gfCNCPoint5[12058] = {X 116.0973, Y 79.9611, Z -7.1667, A 0.000, B 0.000, C 0.000 }
gfCNCPoint5[12059] = {X 117.8219, Y 79.1683, Z -7.1667, A 0.000, B 0.000, C 0.000 }
gfCNCPoint5[12060] = {X 119.6162, Y 78.5490, Z -7.1667, A 0.000, B 0.000, C 0.000 }
gfCNCPoint5[12061] = {X 137.8560, Y 58.5204, Z -7.1667, A 0.000, B 0.000, C 0.000 }
gfCNCPoint5[12062] = {X 136.5214, Y 57.9299, Z -7.1667, A 0.000, B 0.000, C 0.000 }
gfCNCPoint5[12063] = {X 135.2529, Y 57.2081, Z -7.1667, A 0.000, B 0.000, C 0.000 }
gfCNCPoint5[12064] = {X 134.0093, Y 56.3192, Z -7.1667, A 0.000, B 0.000, C 0.000 }
gfCNCPoint5[12065] = {X 132.8663, Y 55.3040, Z -7.1667, A 0.000, B 0.000, C 0.000 }
gfCNCPoint5[12066] = {X 131.8367, Y 54.1741, Z -7.1667, A 0.000, B 0.000, C 0.000 }
gfCNCPoint5[12067] = {X 130.9319, Y 52.9419, Z -7.1667, A 0.000, B 0.000, C 0.000 }
gfCNCPoint5[12068] = {X 130.2147, Y 51.7225, Z -7.1667, A 0.000, B 0.000, C 0.000 }
gfCNCPoint5[12069] = {X 129.6199, Y 50.4390, Z -7.1667, A 0.000, B 0.000, C 0.000 }
gfCNCPoint5[12070] = {X 129.1532, Y 49.1035, Z -7.1667, A 0.000, B 0.000, C 0.000 }
gfCNCPoint5[12071] = {X 128.6036, Y 50.3877, Z -7.1667, A 0.000, B 0.000, C 0.000 }
gfCNCPoint5[12072] = {X 127.9093, Y 51.5998, Z -7.1667, A 0.000, B 0.000, C 0.000 }
gfCNCPoint5[12073] = {X 127.0798, Y 52.7237, Z -7.1667, A 0.000, B 0.000, C 0.000 }
gfCNCPoint5[12074] = {X 126.0417, Y 53.8239, Z -7.1667, A 0.000, B 0.000, C 0.000 }
gfCNCPoint5[12075] = {X 124.8743, Y 54.7858, Z -7.1667, A 0.000, B 0.000, C 0.000 }
gfCNCPoint5[12076] = {X 123.5958, Y 55.5942, Z -7.1667, A 0.000, B 0.000, C 0.000 }
gfCNCPoint5[12077] = {X 122.2263, Y 56.2365, Z -7.1667, A 0.000, B 0.000, C 0.000 }
gfCNCPoint5[12078] = {X 120.7872, Y 56.7027, Z -7.1667, A 0.000, B 0.000, C 0.000 }
gfCNCPoint5[12079] = {X 119.3012, Y 56.9853, Z -7.1667, A 0.000, B 0.000, C 0.000 }
gfCNCPoint5[12080] = {X 117.7916, Y 57.0800, Z -7.1667, A 0.000, B 0.000, C 0.000 }
gfCNCPoint5[12081] = {X 111.9185, Y 57.0800, Z -7.1667, A 0.000, B 0.000, C 0.000 }
gfCNCPoint5[12082] = {X 111.7011, Y 57.0780, Z -7.1667, A 0.000, B 0.000, C 0.000 }
gfCNCPoint5[12083] = {X 111.4838, Y 57.0722, Z -7.1667, A 0.000, B 0.000, C 0.000 }
gfCNCPoint5[12084] = {X 111.5702, Y 54.6737, Z -7.1667, A 0.000, B 0.000, C 0.000 }
gfCNCPoint5[12085] = {X 110.3801, Y 54.5570, Z -7.1667, A 0.000, B 0.000, C 0.000 }
gfCNCPoint5[12086] = {X 109.2135, Y 54.2944, Z -7.1667, A 0.000, B 0.000, C 0.000 }
gfCNCPoint5[12087] = {X 108.0882, Y 53.8899, Z -7.1667, A 0.000, B 0.000, C 0.000 }
gfCNCPoint5[12088] = {X 107.0213, Y 53.3498, Z -7.1667, A 0.000, B 0.000, C 0.000 }
gfCNCPoint5[12089] = {X 106.6480, Y 53.5578, Z -7.1667, A 0.000, B 0.000, C 0.000 }
gfCNCPoint5[12090] = {X 106.2658, Y 53.7492, Z -7.1667, A 0.000, B 0.000, C 0.000 }
gfCNCPoint5[12091] = {X 105.0149, Y 54.2383, Z -7.1667, A 0.000, B 0.000, C 0.000 }
gfCNCPoint5[12092] = {X 103.7084, Y 54.5495, Z -7.1667, A 0.000, B 0.000, C 0.000 }
gfCNCPoint5[12093] = {X 102.3713, Y 54.6768, Z -7.1667, A 0.000, B 0.000, C 0.000 }
gfCNCPoint5[12094] = {X 101.0295, Y 54.6179, Z -7.1667, A 0.000, B 0.000, C 0.000 }
gfCNCPoint5[12095] = {X 99.7088, Y 54.3738, Z -7.1667, A 0.000, B 0.000, C 0.000 }
gfCNCPoint5[12096] = {X 98.4345, Y 53.9493, Z -7.1667, A 0.000, B 0.000, C 0.000 }
gfCNCPoint5[12097] = {X 97.2313, Y 53.3524, Z -7.1667, A 0.000, B 0.000, C 0.000 }
gfCNCPoint5[12098] = {X 96.0852, Y 53.9255, Z -7.1667, A 0.000, B 0.000, C 0.000 }
gfCNCPoint5[12099] = {X 94.8734, Y 54.3422, Z -7.1667, A 0.000, B 0.000, C 0.000 }
gfCNCPoint5[12100] = {X 93.6172, Y 54.5952, Z -7.1667, A 0.000, B 0.000, C 0.000 }
gfCNCPoint5[12101] = {X 92.3385, Y 54.6800, Z -7.1667, A 0.000, B 0.000, C 0.000 }
gfCNCPoint5[12102] = {X 85.8951, Y 54.6800, Z -7.1667, A 0.000, B 0.000, C 0.000 }
gfCNCPoint5[12103] = {X 84.6159, Y 54.5951, Z -7.1667, A 0.000, B 0.000, C 0.000 }
gfCNCPoint5[12104] = {X 83.3592, Y 54.3419, Z -7.1667, A 0.000, B 0.000, C 0.000 }
gfCNCPoint5[12105] = {X 82.1469, Y 53.9249, Z -7.1667, A 0.000, B 0.000, C 0.000 }
gfCNCPoint5[12106] = {X 81.0644, Y 55.1572, Z -7.1667, A 0.000, B 0.000, C 0.000 }
gfCNCPoint5[12107] = {X 79.8495, Y 56.2591, Z -7.1667, A 0.000, B 0.000, C 0.000 }
gfCNCPoint5[12108] = {X 78.5178, Y 57.2166, Z -7.1667, A 0.000, B 0.000, C 0.000 }
gfCNCPoint5[12109] = {X 77.0863, Y 58.0174, Z -7.1667, A 0.000, B 0.000, C 0.000 }
gfCNCPoint5[12110] = {X 75.5734, Y 58.6511, Z -7.1667, A 0.000, B 0.000, C 0.000 }
gfCNCPoint5[12111] = {X 73.9986, Y 59.1096, Z -7.1667, A 0.000, B 0.000, C 0.000 }
gfCNCPoint5[12112] = {X 72.3820, Y 59.3871, Z -7.1667, A 0.000, B 0.000, C 0.000 }
gfCNCPoint5[12113] = {X 70.7445, Y 59.4800, Z -7.1667, A 0.000, B 0.000, C 0.000 }
gfCNCPoint5[12114] = {X 64.1851, Y 59.4800, Z -7.1667, A 0.000, B 0.000, C 0.000 }
gfCNCPoint5[12115] = {X 62.4203, Y 59.3720, Z -7.1667, A 0.000, B 0.000, C 0.000 }
gfCNCPoint5[12116] = {X 60.6818, Y 59.0498, Z -7.1667, A 0.000, B 0.000, C 0.000 }
gfCNCPoint5[12117] = {X 58.9955, Y 58.5181, Z -7.1667, A 0.000, B 0.000, C 0.000 }
gfCNCPoint5[12118] = {X 57.3866, Y 57.7848, Z -7.1667, A 0.000, B 0.000, C 0.000 }
gfCNCPoint5[12119] = {X 55.8790, Y 56.8608, Z -7.1667, A 0.000, B 0.000, C 0.000 }
gfCNCPoint5[12120] = {X 54.3715, Y 57.7848, Z -7.1667, A 0.000, B 0.000, C 0.000 }
gfCNCPoint5[12121] = {X 52.7626, Y 58.5181, Z -7.1667, A 0.000, B 0.000, C 0.000 }
gfCNCPoint5[12122] = {X 51.0763, Y 59.0498, Z -7.1667, A 0.000, B 0.000, C 0.000 }
gfCNCPoint5[12123] = {X 49.3378, Y 59.3720, Z -7.1667, A 0.000, B 0.000, C 0.000 }
gfCNCPoint5[12124] = {X 47.5729, Y 59.4800, Z -7.1667, A 0.000, B 0.000, C 0.000 }
gfCNCPoint5[12125] = {X 40.6393, Y 59.4800, Z -7.1667, A 0.000, B 0.000, C 0.000 }
gfCNCPoint5[12126] = {X 38.9799, Y 59.3846, Z -7.1667, A 0.000, B 0.000, C 0.000 }
gfCNCPoint5[12127] = {X 37.3423, Y 59.0996, Z -7.1667, A 0.000, B 0.000, C 0.000 }
gfCNCPoint5[12128] = {X 35.7482, Y 58.6289, Z -7.1667, A 0.000, B 0.000, C 0.000 }
gfCNCPoint5[12129] = {X 34.0334, Y 59.4877, Z -7.1667, A 0.000, B 0.000, C 0.000 }
gfCNCPoint5[12130] = {X 32.2400, Y 60.1674, Z -7.1667, A 0.000, B 0.000, C 0.000 }
gfCNCPoint5[12131] = {X 30.3868, Y 60.6610, Z -7.1667, A 0.000, B 0.000, C 0.000 }
gfCNCPoint5[12132] = {X 28.4929, Y 60.9633, Z -7.1667, A 0.000, B 0.000, C 0.000 }
gfCNCPoint5[12133] = {X 26.3340, Y 61.8578, Z -7.1667, A 0.000, B 0.000, C 0.000 }
gfCNCPoint5[12134] = {X 24.1304, Y 62.6356, Z -7.1667, A 0.000, B 0.000, C 0.000 }
gfCNCPoint5[12135] = {X 21.7252, Y 63.3378, Z -7.1667, A 0.000, B 0.000, C 0.000 }
gfCNCPoint5[12136] = {X 19.2782, Y 63.8767, Z -7.1667, A 0.000, B 0.000, C 0.000 }
gfCNCPoint5[12137] = {X 16.8005, Y 64.2498, Z -7.1667, A 0.000, B 0.000, C 0.000 }
gfCNCPoint5[12138] = {X 14.3033, Y 64.4554, Z -7.1667, A 0.000, B 0.000, C 0.000 }
gfCNCPoint5[12139] = {X 14.3033, Y 85.6951, Z -7.1667, A 0.000, B 0.000, C 0.000 }
gfCNCPoint5[12140] = {X 112.5225, Y 85.6951, Z -7.1667, A 0.000, B 0.000, C 0.000 }
gfCNCPoint5[12141] = {X 113.9417, Y 84.3100, Z -7.1667, A 0.000, B 0.000, C 0.000 }
gfCNCPoint5[12142] = {X 115.5135, Y 83.1008, Z -7.1667, A 0.000, B 0.000, C 0.000 }
gfCNCPoint5[12143] = {X 117.2162, Y 82.0843, Z -7.1667, A 0.000, B 0.000, C 0.000 }
gfCNCPoint5[12144] = {X 119.0264, Y 81.2746, Z -7.1667, A 0.000, B 0.000, C 0.000 }
gfCNCPoint5[12145] = {X 120.9191, Y 80.6827, Z -7.1667, A 0.000, B 0.000, C 0.000 }
gfCNCPoint5[12146] = {X 142.4280, Y 57.0645, Z -7.1667, A 0.000, B 0.000, C 0.000 }
gfCNCPoint5[12147] = {X 141.1651, Y 56.9337, Z -7.1667, A 0.000, B 0.000, C 0.000 }
gfCNCPoint5[12148] = {X 139.9229, Y 56.6710, Z -7.1667, A 0.000, B 0.000, C 0.000 }
gfCNCPoint5[12149] = {X 138.7152, Y 56.2794, Z -7.1667, A 0.000, B 0.000, C 0.000 }
gfCNCPoint5[12150] = {X 137.2783, Y 55.6176, Z -7.1667, A 0.000, B 0.000, C 0.000 }
gfCNCPoint5[12151] = {X 135.9402, Y 54.7737, Z -7.1667, A 0.000, B 0.000, C 0.000 }
gfCNCPoint5[12152] = {X 134.7239, Y 53.7622, Z -7.1667, A 0.000, B 0.000, C 0.000 }
gfCNCPoint5[12153] = {X 133.6502, Y 52.6004, Z -7.1667, A 0.000, B 0.000, C 0.000 }
gfCNCPoint5[12154] = {X 132.7375, Y 51.3082, Z -7.1667, A 0.000, B 0.000, C 0.000 }
gfCNCPoint5[12155] = {X 132.0015, Y 49.9079, Z -7.1667, A 0.000, B 0.000, C 0.000 }
gfCNCPoint5[12156] = {X 131.4549, Y 48.4234, Z -7.1667, A 0.000, B 0.000, C 0.000 }
gfCNCPoint5[12157] = {X 131.1845, Y 47.3200, Z -7.1667, A 0.000, B 0.000, C 0.000 }
gfCNCPoint5[12158] = {X 131.0190, Y 46.1961, Z -7.1667, A 0.000, B 0.000, C 0.000 }
gfCNCPoint5[12159] = {X 130.9598, Y 45.0616, Z -7.1667, A 0.000, B 0.000, C 0.000 }
gfCNCPoint5[12160] = {X 130.9601, Y 44.0979, Z -7.1667, A 0.000, B 0.000, C 0.000 }
gfCNCPoint5[12161] = {X 131.0921, Y 42.4244, Z -7.1667, A 0.000, B 0.000, C 0.000 }
gfCNCPoint5[12162] = {X 131.4548, Y 40.7854, Z -7.1667, A 0.000, B 0.000, C 0.000 }
gfCNCPoint5[12163] = {X 133.7565, Y 41.4655, Z -7.1667, A 0.000, B 0.000, C 0.000 }
gfCNCPoint5[12164] = {X 134.2330, Y 40.1906, Z -7.1667, A 0.000, B 0.000, C 0.000 }
gfCNCPoint5[12165] = {X 134.8836, Y 38.9952, Z -7.1667, A 0.000, B 0.000, C 0.000 }
gfCNCPoint5[12166] = {X 134.8836, Y 27.0854, Z -7.1667, A 0.000, B 0.000, C 0.000 }
gfCNCPoint5[12167] = {X 134.3931, Y 27.1259, Z -7.1667, A 0.000, B 0.000, C 0.000 }
gfCNCPoint5[12168] = {X 133.9011, Y 27.1414, Z -7.1667, A 0.000, B 0.000, C 0.000 }
gfCNCPoint5[12169] = {X 133.2006, Y 27.1415, Z -7.1667, A 0.000, B 0.000, C 0.000 }
gfCNCPoint5[12170] = {X 131.9568, Y 27.0613, Z -7.1667, A 0.000, B 0.000, C 0.000 }
gfCNCPoint5[12171] = {X 130.7335, Y 26.8219, Z -7.1667, A 0.000, B 0.000, C 0.000 }
gfCNCPoint5[12172] = {X 129.5511, Y 26.4272, Z -7.1667, A 0.000, B 0.000, C 0.000 }
gfCNCPoint5[12173] = {X 128.4293, Y 25.8839, Z -7.1667, A 0.000, B 0.000, C 0.000 }
gfCNCPoint5[12174] = {X 127.3866, Y 25.2010, Z -7.1667, A 0.000, B 0.000, C 0.000 }
gfCNCPoint5[12175] = {X 126.3459, Y 24.2964, Z -7.1667, A 0.000, B 0.000, C 0.000 }
gfCNCPoint5[12176] = {X 125.4444, Y 23.2532, Z -7.1667, A 0.000, B 0.000, C 0.000 }
gfCNCPoint5[12177] = {X 124.7002, Y 22.0924, Z -7.1667, A 0.000, B 0.000, C 0.000 }
gfCNCPoint5[12178] = {X 124.1285, Y 20.8377, Z -7.1667, A 0.000, B 0.000, C 0.000 }
gfCNCPoint5[12179] = {X 123.7409, Y 19.5145, Z -7.1667, A 0.000, B 0.000, C 0.000 }
gfCNCPoint5[12180] = {X 123.5451, Y 18.1497, Z -7.1667, A 0.000, B 0.000, C 0.000 }
gfCNCPoint5[12181] = {X 123.5450, Y 39.7482, Z -7.1667, A 0.000, B 0.000, C 0.000 }
gfCNCPoint5[12182] = {X 124.1931, Y 40.7420, Z -7.1667, A 0.000, B 0.000, C 0.000 }
gfCNCPoint5[12183] = {X 124.6712, Y 41.8278, Z -7.1667, A 0.000, B 0.000, C 0.000 }
gfCNCPoint5[12184] = {X 124.9666, Y 42.9769, Z -7.1667, A 0.000, B 0.000, C 0.000 }
gfCNCPoint5[12185] = {X 125.0714, Y 44.1587, Z -7.1667, A 0.000, B 0.000, C 0.000 }
gfCNCPoint5[12186] = {X 125.0716, Y 45.0000, Z -7.1667, A 0.000, B 0.000, C 0.000 }
gfCNCPoint5[12187] = {X 124.9610, Y 46.2642, Z -7.1667, A 0.000, B 0.000, C 0.000 }
gfCNCPoint5[12188] = {X 124.6325, Y 47.4899, Z -7.1667, A 0.000, B 0.000, C 0.000 }
gfCNCPoint5[12189] = {X 124.0962, Y 48.6400, Z -7.1667, A 0.000, B 0.000, C 0.000 }
gfCNCPoint5[12190] = {X 123.3684, Y 49.6795, Z -7.1667, A 0.000, B 0.000, C 0.000 }
gfCNCPoint5[12191] = {X 122.4711, Y 50.5768, Z -7.1667, A 0.000, B 0.000, C 0.000 }
gfCNCPoint5[12192] = {X 121.4316, Y 51.3047, Z -7.1667, A 0.000, B 0.000, C 0.000 }
gfCNCPoint5[12193] = {X 120.2815, Y 51.8410, Z -7.1667, A 0.000, B 0.000, C 0.000 }
gfCNCPoint5[12194] = {X 119.0557, Y 52.1694, Z -7.1667, A 0.000, B 0.000, C 0.000 }
gfCNCPoint5[12195] = {X 117.7916, Y 52.2800, Z -7.1667, A 0.000, B 0.000, C 0.000 }
gfCNCPoint5[12196] = {X 111.9185, Y 52.2800, Z -7.1667, A 0.000, B 0.000, C 0.000 }
gfCNCPoint5[12197] = {X 110.8481, Y 52.2009, Z -7.1667, A 0.000, B 0.000, C 0.000 }
gfCNCPoint5[12198] = {X 109.8009, Y 51.9652, Z -7.1667, A 0.000, B 0.000, C 0.000 }
gfCNCPoint5[12199] = {X 108.7998, Y 51.5782, Z -7.1667, A 0.000, B 0.000, C 0.000 }
gfCNCPoint5[12200] = {X 107.8665, Y 51.0481, Z -7.1667, A 0.000, B 0.000, C 0.000 }
gfCNCPoint5[12201] = {X 107.0213, Y 50.3866, Z -7.1667, A 0.000, B 0.000, C 0.000 }
gfCNCPoint5[12202] = {X 106.1743, Y 51.0493, Z -7.1667, A 0.000, B 0.000, C 0.000 }
gfCNCPoint5[12203] = {X 105.2389, Y 51.5800, Z -7.1667, A 0.000, B 0.000, C 0.000 }
gfCNCPoint5[12204] = {X 104.0917, Y 52.0091, Z -7.1667, A 0.000, B 0.000, C 0.000 }
gfCNCPoint5[12205] = {X 102.8887, Y 52.2397, Z -7.1667, A 0.000, B 0.000, C 0.000 }
gfCNCPoint5[12206] = {X 101.6641, Y 52.2655, Z -7.1667, A 0.000, B 0.000, C 0.000 }
gfCNCPoint5[12207] = {X 100.4526, Y 52.0855, Z -7.1667, A 0.000, B 0.000, C 0.000 }
gfCNCPoint5[12208] = {X 99.2883, Y 51.7050, Z -7.1667, A 0.000, B 0.000, C 0.000 }
gfCNCPoint5[12209] = {X 98.2043, Y 51.1347, Z -7.1667, A 0.000, B 0.000, C 0.000 }
gfCNCPoint5[12210] = {X 97.2313, Y 50.3907, Z -7.1667, A 0.000, B 0.000, C 0.000 }
gfCNCPoint5[12211] = {X 96.3865, Y 51.0508, Z -7.1667, A 0.000, B 0.000, C 0.000 }
gfCNCPoint5[12212] = {X 95.4539, Y 51.5797, Z -7.1667, A 0.000, B 0.000, C 0.000 }
gfCNCPoint5[12213] = {X 94.4538, Y 51.9659, Z -7.1667, A 0.000, B 0.000, C 0.000 }
gfCNCPoint5[12214] = {X 93.4078, Y 52.2011, Z -7.1667, A 0.000, B 0.000, C 0.000 }
gfCNCPoint5[12215] = {X 92.3385, Y 52.2800, Z -7.1667, A 0.000, B 0.000, C 0.000 }
gfCNCPoint5[12216] = {X 85.8951, Y 52.2800, Z -7.1667, A 0.000, B 0.000, C 0.000 }
gfCNCPoint5[12217] = {X 84.6852, Y 52.1788, Z -7.1667, A 0.000, B 0.000, C 0.000 }
gfCNCPoint5[12218] = {X 83.5090, Y 51.8779, Z -7.1667, A 0.000, B 0.000, C 0.000 }
gfCNCPoint5[12219] = {X 82.3992, Y 51.3857, Z -7.1667, A 0.000, B 0.000, C 0.000 }
gfCNCPoint5[12220] = {X 81.3866, Y 50.7159, Z -7.1667, A 0.000, B 0.000, C 0.000 }
gfCNCPoint5[12221] = {X 80.5223, Y 52.0937, Z -7.1667, A 0.000, B 0.000, C 0.000 }
gfCNCPoint5[12222] = {X 79.4808, Y 53.3429, Z -7.1667, A 0.000, B 0.000, C 0.000 }
gfCNCPoint5[12223] = {X 78.2809, Y 54.4408, Z -7.1667, A 0.000, B 0.000, C 0.000 }
gfCNCPoint5[12224] = {X 76.9444, Y 55.3676, Z -7.1667, A 0.000, B 0.000, C 0.000 }
gfCNCPoint5[12225] = {X 75.4955, Y 56.1065, Z -7.1667, A 0.000, B 0.000, C 0.000 }
gfCNCPoint5[12226] = {X 73.9605, Y 56.6440, Z -7.1667, A 0.000, B 0.000, C 0.000 }
gfCNCPoint5[12227] = {X 72.3672, Y 56.9705, Z -7.1667, A 0.000, B 0.000, C 0.000 }
gfCNCPoint5[12228] = {X 70.7445, Y 57.0800, Z -7.1667, A 0.000, B 0.000, C 0.000 }
gfCNCPoint5[12229] = {X 64.1851, Y 57.0800, Z -7.1667, A 0.000, B 0.000, C 0.000 }
gfCNCPoint5[12230] = {X 62.6628, Y 56.9837, Z -7.1667, A 0.000, B 0.000, C 0.000 }
gfCNCPoint5[12231] = {X 61.1646, Y 56.6963, Z -7.1667, A 0.000, B 0.000, C 0.000 }
gfCNCPoint5[12232] = {X 59.7147, Y 56.2224, Z -7.1667, A 0.000, B 0.000, C 0.000 }
gfCNCPoint5[12233] = {X 58.3360, Y 55.5695, Z -7.1667, A 0.000, B 0.000, C 0.000 }
gfCNCPoint5[12234] = {X 57.0507, Y 54.7481, Z -7.1667, A 0.000, B 0.000, C 0.000 }
gfCNCPoint5[12235] = {X 55.8790, Y 53.7713, Z -7.1667, A 0.000, B 0.000, C 0.000 }
gfCNCPoint5[12236] = {X 54.7074, Y 54.7481, Z -7.1667, A 0.000, B 0.000, C 0.000 }
gfCNCPoint5[12237] = {X 53.4220, Y 55.5695, Z -7.1667, A 0.000, B 0.000, C 0.000 }
gfCNCPoint5[12238] = {X 52.0434, Y 56.2224, Z -7.1667, A 0.000, B 0.000, C 0.000 }
gfCNCPoint5[12239] = {X 50.5934, Y 56.6963, Z -7.1667, A 0.000, B 0.000, C 0.000 }
gfCNCPoint5[12240] = {X 49.0953, Y 56.9837, Z -7.1667, A 0.000, B 0.000, C 0.000 }
gfCNCPoint5[12241] = {X 47.5729, Y 57.0800, Z -7.1667, A 0.000, B 0.000, C 0.000 }
gfCNCPoint5[12242] = {X 40.6393, Y 57.0800, Z -7.1667, A 0.000, B 0.000, C 0.000 }
gfCNCPoint5[12243] = {X 39.3239, Y 57.0082, Z -7.1667, A 0.000, B 0.000, C 0.000 }
gfCNCPoint5[12244] = {X 38.0241, Y 56.7935, Z -7.1667, A 0.000, B 0.000, C 0.000 }
gfCNCPoint5[12245] = {X 36.7554, Y 56.4386, Z -7.1667, A 0.000, B 0.000, C 0.000 }
gfCNCPoint5[12246] = {X 35.5329, Y 55.9476, Z -7.1667, A 0.000, B 0.000, C 0.000 }
gfCNCPoint5[12247] = {X 34.1220, Y 56.7828, Z -7.1667, A 0.000, B 0.000, C 0.000 }
gfCNCPoint5[12248] = {X 32.6348, Y 57.4730, Z -7.1667, A 0.000, B 0.000, C 0.000 }
gfCNCPoint5[12249] = {X 31.0862, Y 58.0113, Z -7.1667, A 0.000, B 0.000, C 0.000 }
gfCNCPoint5[12250] = {X 29.4916, Y 58.3925, Z -7.1667, A 0.000, B 0.000, C 0.000 }
gfCNCPoint5[12251] = {X 27.8669, Y 58.6126, Z -7.1667, A 0.000, B 0.000, C 0.000 }
gfCNCPoint5[12252] = {X 25.6520, Y 59.5485, Z -7.1667, A 0.000, B 0.000, C 0.000 }
gfCNCPoint5[12253] = {X 23.3865, Y 60.3538, Z -7.1667, A 0.000, B 0.000, C 0.000 }
gfCNCPoint5[12254] = {X 21.1469, Y 61.0085, Z -7.1667, A 0.000, B 0.000, C 0.000 }
gfCNCPoint5[12255] = {X 18.8685, Y 61.5117, Z -7.1667, A 0.000, B 0.000, C 0.000 }
gfCNCPoint5[12256] = {X 16.5615, Y 61.8614, Z -7.1667, A 0.000, B 0.000, C 0.000 }
gfCNCPoint5[12257] = {X 14.2363, Y 62.0558, Z -7.1667, A 0.000, B 0.000, C 0.000 }
gfCNCPoint5[12258] = {X 11.9033, Y 62.0941, Z -7.1667, A 0.000, B 0.000, C 0.000 }
gfCNCPoint5[12259] = {X 11.9033, Y 88.0951, Z -7.1667, A 0.000, B 0.000, C 0.000 }
gfCNCPoint5[12260] = {X 113.6322, Y 88.0951, Z -7.1667, A 0.000, B 0.000, C 0.000 }
gfCNCPoint5[12261] = {X 114.7654, Y 86.8204, Z -7.1667, A 0.000, B 0.000, C 0.000 }
gfCNCPoint5[12262] = {X 116.0407, Y 85.6877, Z -7.1667, A 0.000, B 0.000, C 0.000 }
gfCNCPoint5[12263] = {X 117.4402, Y 84.7128, Z -7.1667, A 0.000, B 0.000, C 0.000 }
gfCNCPoint5[12264] = {X 118.9448, Y 83.9093, Z -7.1667, A 0.000, B 0.000, C 0.000 }
gfCNCPoint5[12265] = {X 120.5333, Y 83.2883, Z -7.1667, A 0.000, B 0.000, C 0.000 }
gfCNCPoint5[12266] = {X 122.1839, Y 82.8584, Z -7.1667, A 0.000, B 0.000, C 0.000 }
gfCNCPoint5[12267] = {X 144.8180, Y 58.0046, Z -7.1667, A 0.000, B 0.000, C 0.000 }
gfCNCPoint5[12268] = {X 144.9145, Y 56.3311, Z -7.1667, A 0.000, B 0.000, C 0.000 }
gfCNCPoint5[12269] = {X 145.2037, Y 54.6800, Z -7.1667, A 0.000, B 0.000, C 0.000 }
gfCNCPoint5[12270] = {X 143.0396, Y 54.6800, Z -7.1667, A 0.000, B 0.000, C 0.000 }
gfCNCPoint5[12271] = {X 142.7945, Y 54.6769, Z -7.1667, A 0.000, B 0.000, C 0.000 }
gfCNCPoint5[12272] = {X 142.5495, Y 54.6676, Z -7.1667, A 0.000, B 0.000, C 0.000 }
gfCNCPoint5[12273] = {X 141.0966, Y 54.4830, Z -7.1667, A 0.000, B 0.000, C 0.000 }
gfCNCPoint5[12274] = {X 139.6882, Y 54.0813, Z -7.1667, A 0.000, B 0.000, C 0.000 }
gfCNCPoint5[12275] = {X 138.3565, Y 53.4718, Z -7.1667, A 0.000, B 0.000, C 0.000 }
gfCNCPoint5[12276] = {X 137.1320, Y 52.6683, Z -7.1667, A 0.000, B 0.000, C 0.000 }
gfCNCPoint5[12277] = {X 136.0427, Y 51.6892, Z -7.1667, A 0.000, B 0.000, C 0.000 }
gfCNCPoint5[12278] = {X 135.1136, Y 50.5571, Z -7.1667, A 0.000, B 0.000, C 0.000 }
gfCNCPoint5[12279] = {X 134.3660, Y 49.2977, Z -7.1667, A 0.000, B 0.000, C 0.000 }
gfCNCPoint5[12280] = {X 133.8169, Y 47.9400, Z -7.1667, A 0.000, B 0.000, C 0.000 }
gfCNCPoint5[12281] = {X 133.4789, Y 46.5149, Z -7.1667, A 0.000, B 0.000, C 0.000 }
gfCNCPoint5[12282] = {X 133.3598, Y 45.0552, Z -7.1667, A 0.000, B 0.000, C 0.000 }
gfCNCPoint5[12283] = {X 133.3601, Y 44.1105, Z -7.1667, A 0.000, B 0.000, C 0.000 }
gfCNCPoint5[12284] = {X 133.4665, Y 42.7743, Z -7.1667, A 0.000, B 0.000, C 0.000 }
gfCNCPoint5[12285] = {X 133.7565, Y 41.4655, Z -7.1667, A 0.000, B 0.000, C 0.000 }
gfCNCPoint5[12286] = {X 136.0581, Y 42.1457, Z -7.1667, A 0.000, B 0.000, C 0.000 }
gfCNCPoint5[12287] = {X 136.3664, Y 41.2990, Z -7.1667, A 0.000, B 0.000, C 0.000 }
gfCNCPoint5[12288] = {X 136.7770, Y 40.4969, Z -7.1667, A 0.000, B 0.000, C 0.000 }
gfCNCPoint5[12289] = {X 137.2836, Y 39.7516, Z -7.1667, A 0.000, B 0.000, C 0.000 }
gfCNCPoint5[12290] = {X 137.2836, Y 23.8768, Z -7.1667, A 0.000, B 0.000, C 0.000 }
gfCNCPoint5[12291] = {X 136.4352, Y 24.2641, Z -7.1667, A 0.000, B 0.000, C 0.000 }
gfCNCPoint5[12292] = {X 135.5443, Y 24.5398, Z -7.1667, A 0.000, B 0.000, C 0.000 }
gfCNCPoint5[12293] = {X 134.6254, Y 24.6993, Z -7.1667, A 0.000, B 0.000, C 0.000 }
gfCNCPoint5[12294] = {X 134.2595, Y 24.7296, Z -7.1667, A 0.000, B 0.000, C 0.000 }
gfCNCPoint5[12295] = {X 133.8926, Y 24.7414, Z -7.1667, A 0.000, B 0.000, C 0.000 }
gfCNCPoint5[12296] = {X 133.2006, Y 24.7415, Z -7.1667, A 0.000, B 0.000, C 0.000 }
gfCNCPoint5[12297] = {X 131.9932, Y 24.6407, Z -7.1667, A 0.000, B 0.000, C 0.000 }
gfCNCPoint5[12298] = {X 130.8192, Y 24.3410, Z -7.1667, A 0.000, B 0.000, C 0.000 }
gfCNCPoint5[12299] = {X 129.7112, Y 23.8507, Z -7.1667, A 0.000, B 0.000, C 0.000 }
gfCNCPoint5[12300] = {X 128.6998, Y 23.1835, Z -7.1667, A 0.000, B 0.000, C 0.000 }
gfCNCPoint5[12301] = {X 127.8131, Y 22.3578, Z -7.1667, A 0.000, B 0.000, C 0.000 }
gfCNCPoint5[12302] = {X 127.0757, Y 21.3964, Z -7.1667, A 0.000, B 0.000, C 0.000 }
gfCNCPoint5[12303] = {X 126.5079, Y 20.3260, Z -7.1667, A 0.000, B 0.000, C 0.000 }
gfCNCPoint5[12304] = {X 126.1255, Y 19.1763, Z -7.1667, A 0.000, B 0.000, C 0.000 }
gfCNCPoint5[12305] = {X 125.9391, Y 17.9791, Z -7.1667, A 0.000, B 0.000, C 0.000 }
gfCNCPoint5[12306] = {X 125.9252, Y 17.7205, Z -7.1667, A 0.000, B 0.000, C 0.000 }
gfCNCPoint5[12307] = {X 125.9206, Y 17.4615, Z -7.1667, A 0.000, B 0.000, C 0.000 }
gfCNCPoint5[12308] = {X 125.9206, Y 10.4835, Z -7.1667, A 0.000, B 0.000, C 0.000 }
gfCNCPoint5[12309] = {X 125.9372, Y 9.9931, Z -7.1667, A 0.000, B 0.000, C 0.000 }
gfCNCPoint5[12310] = {X 125.9867, Y 9.5049, Z -7.1667, A 0.000, B 0.000, C 0.000 }
gfCNCPoint5[12311] = {X 121.8685, Y 9.5049, Z -7.1667, A 0.000, B 0.000, C 0.000 }
gfCNCPoint5[12312] = {X 122.3090, Y 10.3409, Z -7.1667, A 0.000, B 0.000, C 0.000 }
gfCNCPoint5[12313] = {X 122.5801, Y 11.2462, Z -7.1667, A 0.000, B 0.000, C 0.000 }
gfCNCPoint5[12314] = {X 122.6716, Y 12.1868, Z -7.1667, A 0.000, B 0.000, C 0.000 }
gfCNCPoint5[12315] = {X 122.6714, Y 13.0237, Z -7.1667, A 0.000, B 0.000, C 0.000 }
gfCNCPoint5[12316] = {X 122.5640, Y 13.9968, Z -7.1667, A 0.000, B 0.000, C 0.000 }
gfCNCPoint5[12317] = {X 122.2647, Y 14.9289, Z -7.1667, A 0.000, B 0.000, C 0.000 }
gfCNCPoint5[12318] = {X 121.7853, Y 15.7824, Z -7.1667, A 0.000, B 0.000, C 0.000 }
gfCNCPoint5[12319] = {X 121.1451, Y 16.5232, Z -7.1667, A 0.000, B 0.000, C 0.000 }
gfCNCPoint5[12320] = {X 121.1450, Y 40.6635, Z -7.1667, A 0.000, B 0.000, C 0.000 }
gfCNCPoint5[12321] = {X 121.7860, Y 41.4054, Z -7.1667, A 0.000, B 0.000, C 0.000 }
gfCNCPoint5[12322] = {X 122.2658, Y 42.2604, Z -7.1667, A 0.000, B 0.000, C 0.000 }
gfCNCPoint5[12323] = {X 122.5649, Y 43.1941, Z -7.1667, A 0.000, B 0.000, C 0.000 }
gfCNCPoint5[12324] = {X 122.6714, Y 44.1688, Z -7.1667, A 0.000, B 0.000, C 0.000 }
gfCNCPoint5[12325] = {X 122.6716, Y 45.0000, Z -7.1667, A 0.000, B 0.000, C 0.000 }
gfCNCPoint5[12326] = {X 122.5778, Y 45.9520, Z -7.1667, A 0.000, B 0.000, C 0.000 }
gfCNCPoint5[12327] = {X 122.3001, Y 46.8675, Z -7.1667, A 0.000, B 0.000, C 0.000 }
gfCNCPoint5[12328] = {X 121.8491, Y 47.7112, Z -7.1667, A 0.000, B 0.000, C 0.000 }
gfCNCPoint5[12329] = {X 121.2423, Y 48.4507, Z -7.1667, A 0.000, B 0.000, C 0.000 }
gfCNCPoint5[12330] = {X 120.5028, Y 49.0576, Z -7.1667, A 0.000, B 0.000, C 0.000 }
gfCNCPoint5[12331] = {X 119.6591, Y 49.5085, Z -7.1667, A 0.000, B 0.000, C 0.000 }
gfCNCPoint5[12332] = {X 118.7436, Y 49.7862, Z -7.1667, A 0.000, B 0.000, C 0.000 }
gfCNCPoint5[12333] = {X 117.7916, Y 49.8800, Z -7.1667, A 0.000, B 0.000, C 0.000 }
gfCNCPoint5[12334] = {X 111.9185, Y 49.8800, Z -7.1667, A 0.000, B 0.000, C 0.000 }
gfCNCPoint5[12335] = {X 111.0234, Y 49.7972, Z -7.1667, A 0.000, B 0.000, C 0.000 }
gfCNCPoint5[12336] = {X 110.1587, Y 49.5517, Z -7.1667, A 0.000, B 0.000, C 0.000 }
gfCNCPoint5[12337] = {X 109.3537, Y 49.1517, Z -7.1667, A 0.000, B 0.000, C 0.000 }
gfCNCPoint5[12338] = {X 108.6357, Y 48.6108, Z -7.1667, A 0.000, B 0.000, C 0.000 }
gfCNCPoint5[12339] = {X 108.0714, Y 48.0024, Z -7.1667, A 0.000, B 0.000, C 0.000 }
gfCNCPoint5[12340] = {X 107.6183, Y 47.3071, Z -7.1667, A 0.000, B 0.000, C 0.000 }
gfCNCPoint5[12341] = {X 107.2895, Y 46.5451, Z -7.1667, A 0.000, B 0.000, C 0.000 }
gfCNCPoint5[12342] = {X 107.0947, Y 45.7384, Z -7.1667, A 0.000, B 0.000, C 0.000 }
gfCNCPoint5[12343] = {X 106.6287, Y 46.8770, Z -7.1667, A 0.000, B 0.000, C 0.000 }
gfCNCPoint5[12344] = {X 106.1131, Y 47.8111, Z -7.1667, A 0.000, B 0.000, C 0.000 }
gfCNCPoint5[12345] = {X 105.4068, Y 48.6108, Z -7.1667, A 0.000, B 0.000, C 0.000 }
gfCNCPoint5[12346] = {X 104.8391, Y 49.0550, Z -7.1667, A 0.000, B 0.000, C 0.000 }
gfCNCPoint5[12347] = {X 104.2121, Y 49.4107, Z -7.1667, A 0.000, B 0.000, C 0.000 }
gfCNCPoint5[12348] = {X 103.3106, Y 49.7335, Z -7.1667, A 0.000, B 0.000, C 0.000 }
gfCNCPoint5[12349] = {X 102.3635, Y 49.8741, Z -7.1667, A 0.000, B 0.000, C 0.000 }
gfCNCPoint5[12350] = {X 101.4071, Y 49.8271, Z -7.1667, A 0.000, B 0.000, C 0.000 }
gfCNCPoint5[12351] = {X 100.4784, Y 49.5941, Z -7.1667, A 0.000, B 0.000, C 0.000 }
gfCNCPoint5[12352] = {X 99.6130, Y 49.1844, Z -7.1667, A 0.000, B 0.000, C 0.000 }
gfCNCPoint5[12353] = {X 98.8443, Y 48.6135, Z -7.1667, A 0.000, B 0.000, C 0.000 }
gfCNCPoint5[12354] = {X 98.1362, Y 47.8127, Z -7.1667, A 0.000, B 0.000, C 0.000 }
gfCNCPoint5[12355] = {X 97.6194, Y 46.8769, Z -7.1667, A 0.000, B 0.000, C 0.000 }
gfCNCPoint5[12356] = {X 97.1600, Y 45.7536, Z -7.1667, A 0.000, B 0.000, C 0.000 }
gfCNCPoint5[12357] = {X 96.9635, Y 46.5570, Z -7.1667, A 0.000, B 0.000, C 0.000 }
gfCNCPoint5[12358] = {X 96.6342, Y 47.3156, Z -7.1667, A 0.000, B 0.000, C 0.000 }
gfCNCPoint5[12359] = {X 96.1814, Y 48.0078, Z -7.1667, A 0.000, B 0.000, C 0.000 }
gfCNCPoint5[12360] = {X 95.6183, Y 48.6135, Z -7.1667, A 0.000, B 0.000, C 0.000 }
gfCNCPoint5[12361] = {X 94.9007, Y 49.1533, Z -7.1667, A 0.000, B 0.000, C 0.000 }
gfCNCPoint5[12362] = {X 94.0964, Y 49.5524, Z -7.1667, A 0.000, B 0.000, C 0.000 }
gfCNCPoint5[12363] = {X 93.2326, Y 49.7974, Z -7.1667, A 0.000, B 0.000, C 0.000 }
gfCNCPoint5[12364] = {X 92.3385, Y 49.8800, Z -7.1667, A 0.000, B 0.000, C 0.000 }
gfCNCPoint5[12365] = {X 85.8951, Y 49.8800, Z -7.1667, A 0.000, B 0.000, C 0.000 }
gfCNCPoint5[12366] = {X 85.0841, Y 49.8121, Z -7.1667, A 0.000, B 0.000, C 0.000 }
gfCNCPoint5[12367] = {X 84.2956, Y 49.6104, Z -7.1667, A 0.000, B 0.000, C 0.000 }
gfCNCPoint5[12368] = {X 83.5517, Y 49.2805, Z -7.1667, A 0.000, B 0.000, C 0.000 }
gfCNCPoint5[12369] = {X 82.8729, Y 48.8316, Z -7.1667, A 0.000, B 0.000, C 0.000 }
gfCNCPoint5[12370] = {X 82.2391, Y 48.2324, Z -7.1667, A 0.000, B 0.000, C 0.000 }
gfCNCPoint5[12371] = {X 81.7221, Y 47.5300, Z -7.1667, A 0.000, B 0.000, C 0.000 }
gfCNCPoint5[12372] = {X 81.3384, Y 46.7467, Z -7.1667, A 0.000, B 0.000, C 0.000 }
gfCNCPoint5[12373] = {X 81.1002, Y 45.9077, Z -7.1667, A 0.000, B 0.000, C 0.000 }
gfCNCPoint5[12374] = {X 81.0152, Y 45.0397, Z -7.1667, A 0.000, B 0.000, C 0.000 }
gfCNCPoint5[12375] = {X 81.0151, Y 44.2044, Z -7.1667, A 0.000, B 0.000, C 0.000 }
gfCNCPoint5[12376] = {X 81.1193, Y 43.2204, Z -7.1667, A 0.000, B 0.000, C 0.000 }
gfCNCPoint5[12377] = {X 81.4177, Y 42.2770, Z -7.1667, A 0.000, B 0.000, C 0.000 }
gfCNCPoint5[12378] = {X 81.8983, Y 41.4120, Z -7.1667, A 0.000, B 0.000, C 0.000 }
gfCNCPoint5[12379] = {X 82.5419, Y 40.6604, Z -7.1667, A 0.000, B 0.000, C 0.000 }
gfCNCPoint5[12380] = {X 82.5418, Y 25.2454, Z -7.1667, A 0.000, B 0.000, C 0.000 }
gfCNCPoint5[12381] = {X 77.7418, Y 25.2455, Z -7.1667, A 0.000, B 0.000, C 0.000 }
gfCNCPoint5[12382] = {X 77.7417, Y 18.1958, Z -7.1667, A 0.000, B 0.000, C 0.000 }
gfCNCPoint5[12383] = {X 77.0776, Y 16.9724, Z -7.1667, A 0.000, B 0.000, C 0.000 }
gfCNCPoint5[12384] = {X 76.5959, Y 15.6664, Z -7.1667, A 0.000, B 0.000, C 0.000 }
gfCNCPoint5[12385] = {X 76.3064, Y 14.3049, Z -7.1667, A 0.000, B 0.000, C 0.000 }
gfCNCPoint5[12386] = {X 74.0412, Y 14.3049, Z -7.1667, A 0.000, B 0.000, C 0.000 }
gfCNCPoint5[12387] = {X 73.9994, Y 14.7000, Z -7.1667, A 0.000, B 0.000, C 0.000 }
gfCNCPoint5[12388] = {X 73.9467, Y 15.0937, Z -7.1667, A 0.000, B 0.000, C 0.000 }
gfCNCPoint5[12389] = {X 77.7418, Y 25.2455, Z -7.1667, A 0.000, B 0.000, C 0.000 }
gfCNCPoint5[12390] = {X 80.1418, Y 25.2455, Z -7.1667, A 0.000, B 0.000, C 0.000 }
gfCNCPoint5[12391] = {X 80.1417, Y 17.4386, Z -7.1667, A 0.000, B 0.000, C 0.000 }
gfCNCPoint5[12392] = {X 79.4938, Y 16.4453, Z -7.1667, A 0.000, B 0.000, C 0.000 }
gfCNCPoint5[12393] = {X 79.0158, Y 15.3599, Z -7.1667, A 0.000, B 0.000, C 0.000 }
gfCNCPoint5[12394] = {X 78.7203, Y 14.2114, Z -7.1667, A 0.000, B 0.000, C 0.000 }
gfCNCPoint5[12395] = {X 78.6153, Y 13.0301, Z -7.1667, A 0.000, B 0.000, C 0.000 }
gfCNCPoint5[12396] = {X 78.6151, Y 12.1868, Z -7.1667, A 0.000, B 0.000, C 0.000 }
gfCNCPoint5[12397] = {X 78.6164, Y 12.0458, Z -7.1667, A 0.000, B 0.000, C 0.000 }
gfCNCPoint5[12398] = {X 78.6205, Y 11.9049, Z -7.1667, A 0.000, B 0.000, C 0.000 }
gfCNCPoint5[12399] = {X 71.6988, Y 11.9049, Z -7.1667, A 0.000, B 0.000, C 0.000 }
gfCNCPoint5[12400] = {X 71.7013, Y 12.0458, Z -7.1667, A 0.000, B 0.000, C 0.000 }
gfCNCPoint5[12401] = {X 71.7021, Y 12.1868, Z -7.1667, A 0.000, B 0.000, C 0.000 }
gfCNCPoint5[12402] = {X 71.7016, Y 13.0911, Z -7.1667, A 0.000, B 0.000, C 0.000 }
gfCNCPoint5[12403] = {X 71.6387, Y 14.2143, Z -7.1667, A 0.000, B 0.000, C 0.000 }
gfCNCPoint5[12404] = {X 71.4716, Y 15.3267, Z -7.1667, A 0.000, B 0.000, C 0.000 }
gfCNCPoint5[12405] = {X 78.9568, Y 35.3497, Z -7.1667, A 0.000, B 0.000, C 0.000 }
gfCNCPoint5[12406] = {X 79.5721, Y 35.9627, Z -7.1667, A 0.000, B 0.000, C 0.000 }
gfCNCPoint5[12407] = {X 80.1418, Y 36.6183, Z -7.1667, A 0.000, B 0.000, C 0.000 }
gfCNCPoint5[12408] = {X 80.1418, Y 25.2455, Z -7.1667, A 0.000, B 0.000, C 0.000 }
gfCNCPoint5[12409] = {X 82.5418, Y 25.2454, Z -7.1667, A 0.000, B 0.000, C 0.000 }
gfCNCPoint5[12410] = {X 82.5417, Y 16.5233, Z -7.1667, A 0.000, B 0.000, C 0.000 }
gfCNCPoint5[12411] = {X 81.9009, Y 15.7818, Z -7.1667, A 0.000, B 0.000, C 0.000 }
gfCNCPoint5[12412] = {X 81.4212, Y 14.9271, Z -7.1667, A 0.000, B 0.000, C 0.000 }
gfCNCPoint5[12413] = {X 81.1220, Y 13.9938, Z -7.1667, A 0.000, B 0.000, C 0.000 }
gfCNCPoint5[12414] = {X 81.0153, Y 13.0196, Z -7.1667, A 0.000, B 0.000, C 0.000 }
gfCNCPoint5[12415] = {X 81.0151, Y 12.1868, Z -7.1667, A 0.000, B 0.000, C 0.000 }
gfCNCPoint5[12416] = {X 81.0160, Y 12.0923, Z -7.1667, A 0.000, B 0.000, C 0.000 }
gfCNCPoint5[12417] = {X 81.0187, Y 11.9978, Z -7.1667, A 0.000, B 0.000, C 0.000 }
gfCNCPoint5[12418] = {X 81.1325, Y 11.1229, Z -7.1667, A 0.000, B 0.000, C 0.000 }
gfCNCPoint5[12419] = {X 81.4019, Y 10.2828, Z -7.1667, A 0.000, B 0.000, C 0.000 }
gfCNCPoint5[12420] = {X 81.8181, Y 9.5049, Z -7.1667, A 0.000, B 0.000, C 0.000 }
gfCNCPoint5[12421] = {X 82.2191, Y 9.7687, Z -7.1667, A 0.000, B 0.000, C 0.000 }
gfCNCPoint5[12422] = {X 82.7660, Y 9.0935, Z -7.1667, A 0.000, B 0.000, C 0.000 }
gfCNCPoint5[12423] = {X 83.4348, Y 8.5389, Z -7.1667, A 0.000, B 0.000, C 0.000 }
gfCNCPoint5[12424] = {X 84.1996, Y 8.1266, Z -7.1667, A 0.000, B 0.000, C 0.000 }
gfCNCPoint5[12425] = {X 85.0305, Y 7.8726, Z -7.1667, A 0.000, B 0.000, C 0.000 }
gfCNCPoint5[12426] = {X 85.8951, Y 7.7868, Z -7.1667, A 0.000, B 0.000, C 0.000 }
gfCNCPoint5[12427] = {X 94.0497, Y 7.7868, Z -7.1667, A 0.000, B 0.000, C 0.000 }
gfCNCPoint5[12428] = {X 95.0288, Y 7.8971, Z -7.1667, A 0.000, B 0.000, C 0.000 }
gfCNCPoint5[12429] = {X 95.9588, Y 8.2226, Z -7.1667, A 0.000, B 0.000, C 0.000 }
gfCNCPoint5[12430] = {X 96.7930, Y 8.7468, Z -7.1667, A 0.000, B 0.000, C 0.000 }
gfCNCPoint5[12431] = {X 97.4897, Y 9.4435, Z -7.1667, A 0.000, B 0.000, C 0.000 }
gfCNCPoint5[12432] = {X 98.0139, Y 10.2777, Z -7.1667, A 0.000, B 0.000, C 0.000 }
gfCNCPoint5[12433] = {X 98.3394, Y 11.2077, Z -7.1667, A 0.000, B 0.000, C 0.000 }
gfCNCPoint5[12434] = {X 98.4497, Y 12.1868, Z -7.1667, A 0.000, B 0.000, C 0.000 }
gfCNCPoint5[12435] = {X 98.4494, Y 13.0233, Z -7.1667, A 0.000, B 0.000, C 0.000 }
gfCNCPoint5[12436] = {X 98.3725, Y 13.7987, Z -7.1667, A 0.000, B 0.000, C 0.000 }
gfCNCPoint5[12437] = {X 98.1599, Y 14.5484, Z -7.1667, A 0.000, B 0.000, C 0.000 }
gfCNCPoint5[12438] = {X 97.8184, Y 15.2488, Z -7.1667, A 0.000, B 0.000, C 0.000 }
gfCNCPoint5[12439] = {X 101.8767, Y 25.3091, Z -7.1667, A 0.000, B 0.000, C 0.000 }
gfCNCPoint5[12440] = {X 105.0408, Y 17.4192, Z -7.1667, A 0.000, B 0.000, C 0.000 }
gfCNCPoint5[12441] = {X 105.9234, Y 15.2218, Z -7.1667, A 0.000, B 0.000, C 0.000 }
gfCNCPoint5[12442] = {X 105.5853, Y 14.5146, Z -7.1667, A 0.000, B 0.000, C 0.000 }
gfCNCPoint5[12443] = {X 105.3781, Y 13.7587, Z -7.1667, A 0.000, B 0.000, C 0.000 }
gfCNCPoint5[12444] = {X 105.3083, Y 12.9780, Z -7.1667, A 0.000, B 0.000, C 0.000 }
gfCNCPoint5[12445] = {X 105.3083, Y 12.1868, Z -7.1667, A 0.000, B 0.000, C 0.000 }
gfCNCPoint5[12446] = {X 105.4186, Y 11.2077, Z -7.1667, A 0.000, B 0.000, C 0.000 }
gfCNCPoint5[12447] = {X 105.7440, Y 10.2777, Z -7.1667, A 0.000, B 0.000, C 0.000 }
gfCNCPoint5[12448] = {X 106.2682, Y 9.4435, Z -7.1667, A 0.000, B 0.000, C 0.000 }
gfCNCPoint5[12449] = {X 106.9649, Y 8.7468, Z -7.1667, A 0.000, B 0.000, C 0.000 }
gfCNCPoint5[12450] = {X 107.7992, Y 8.2226, Z -7.1667, A 0.000, B 0.000, C 0.000 }
gfCNCPoint5[12451] = {X 108.7292, Y 7.8971, Z -7.1667, A 0.000, B 0.000, C 0.000 }
gfCNCPoint5[12452] = {X 109.7083, Y 7.7868, Z -7.1667, A 0.000, B 0.000, C 0.000 }
gfCNCPoint5[12453] = {X 117.7916, Y 7.7868, Z -7.1667, A 0.000, B 0.000, C 0.000 }
gfCNCPoint5[12454] = {X 118.7707, Y 7.8971, Z -7.1667, A 0.000, B 0.000, C 0.000 }
gfCNCPoint5[12455] = {X 119.7007, Y 8.2226, Z -7.1667, A 0.000, B 0.000, C 0.000 }
gfCNCPoint5[12456] = {X 120.5349, Y 8.7468, Z -7.1667, A 0.000, B 0.000, C 0.000 }
gfCNCPoint5[12457] = {X 121.2316, Y 9.4435, Z -7.1667, A 0.000, B 0.000, C 0.000 }
gfCNCPoint5[12458] = {X 121.7558, Y 10.2777, Z -7.1667, A 0.000, B 0.000, C 0.000 }
gfCNCPoint5[12459] = {X 122.0813, Y 11.2077, Z -7.1667, A 0.000, B 0.000, C 0.000 }
gfCNCPoint5[12460] = {X 122.1916, Y 12.1868, Z -7.1667, A 0.000, B 0.000, C 0.000 }
gfCNCPoint5[12461] = {X 122.1913, Y 13.0233, Z -7.1667, A 0.000, B 0.000, C 0.000 }
gfCNCPoint5[12462] = {X 122.0831, Y 13.9490, Z -7.1667, A 0.000, B 0.000, C 0.000 }
gfCNCPoint5[12463] = {X 121.7823, Y 14.8311, Z -7.1667, A 0.000, B 0.000, C 0.000 }
gfCNCPoint5[12464] = {X 121.3025, Y 15.6301, Z -7.1667, A 0.000, B 0.000, C 0.000 }
gfCNCPoint5[12465] = {X 120.6651, Y 16.3101, Z -7.1667, A 0.000, B 0.000, C 0.000 }
gfCNCPoint5[12466] = {X 120.6650, Y 40.8770, Z -7.1667, A 0.000, B 0.000, C 0.000 }
gfCNCPoint5[12467] = {X 120.6784, Y 40.8882, Z -7.1667, A 0.000, B 0.000, C 0.000 }
gfCNCPoint5[12468] = {X 121.3172, Y 41.5763, Z -7.1667, A 0.000, B 0.000, C 0.000 }
gfCNCPoint5[12469] = {X 121.7955, Y 42.3843, Z -7.1667, A 0.000, B 0.000, C 0.000 }
gfCNCPoint5[12470] = {X 122.0914, Y 43.2753, Z -7.1667, A 0.000, B 0.000, C 0.000 }
gfCNCPoint5[12471] = {X 122.1916, Y 44.2089, Z -7.1667, A 0.000, B 0.000, C 0.000 }
gfCNCPoint5[12472] = {X 122.1916, Y 45.0000, Z -7.1667, A 0.000, B 0.000, C 0.000 }
gfCNCPoint5[12473] = {X 122.0813, Y 45.9791, Z -7.1667, A 0.000, B 0.000, C 0.000 }
gfCNCPoint5[12474] = {X 121.7558, Y 46.9091, Z -7.1667, A 0.000, B 0.000, C 0.000 }
gfCNCPoint5[12475] = {X 121.2316, Y 47.7434, Z -7.1667, A 0.000, B 0.000, C 0.000 }
gfCNCPoint5[12476] = {X 120.5349, Y 48.4401, Z -7.1667, A 0.000, B 0.000, C 0.000 }
gfCNCPoint5[12477] = {X 119.7007, Y 48.9643, Z -7.1667, A 0.000, B 0.000, C 0.000 }
gfCNCPoint5[12478] = {X 118.7707, Y 49.2897, Z -7.1667, A 0.000, B 0.000, C 0.000 }
gfCNCPoint5[12479] = {X 117.7916, Y 49.4000, Z -7.1667, A 0.000, B 0.000, C 0.000 }
gfCNCPoint5[12480] = {X 111.9185, Y 49.4000, Z -7.1667, A 0.000, B 0.000, C 0.000 }
gfCNCPoint5[12481] = {X 110.9394, Y 49.2897, Z -7.1667, A 0.000, B 0.000, C 0.000 }
gfCNCPoint5[12482] = {X 110.0094, Y 48.9643, Z -7.1667, A 0.000, B 0.000, C 0.000 }
gfCNCPoint5[12483] = {X 109.1751, Y 48.4401, Z -7.1667, A 0.000, B 0.000, C 0.000 }
gfCNCPoint5[12484] = {X 108.4784, Y 47.7433, Z -7.1667, A 0.000, B 0.000, C 0.000 }
gfCNCPoint5[12485] = {X 107.9542, Y 46.9091, Z -7.1667, A 0.000, B 0.000, C 0.000 }
gfCNCPoint5[12486] = {X 107.6288, Y 45.9791, Z -7.1667, A 0.000, B 0.000, C 0.000 }
gfCNCPoint5[12487] = {X 107.5185, Y 45.0000, Z -7.1667, A 0.000, B 0.000, C 0.000 }
gfCNCPoint5[12488] = {X 107.5185, Y 44.1771, Z -7.1667, A 0.000, B 0.000, C 0.000 }
gfCNCPoint5[12489] = {X 107.5545, Y 43.6264, Z -7.1667, A 0.000, B 0.000, C 0.000 }
gfCNCPoint5[12490] = {X 107.6618, Y 43.0851, Z -7.1667, A 0.000, B 0.000, C 0.000 }
gfCNCPoint5[12491] = {X 106.1856, Y 46.6923, Z -7.1667, A 0.000, B 0.000, C 0.000 }
gfCNCPoint5[12492] = {X 105.8087, Y 47.4049, Z -7.1667, A 0.000, B 0.000, C 0.000 }
gfCNCPoint5[12493] = {X 105.3081, Y 48.0367, Z -7.1667, A 0.000, B 0.000, C 0.000 }
gfCNCPoint5[12494] = {X 104.7006, Y 48.5667, Z -7.1667, A 0.000, B 0.000, C 0.000 }
gfCNCPoint5[12495] = {X 104.0067, Y 48.9769, Z -7.1667, A 0.000, B 0.000, C 0.000 }
gfCNCPoint5[12496] = {X 103.0414, Y 49.3033, Z -7.1667, A 0.000, B 0.000, C 0.000 }
gfCNCPoint5[12497] = {X 102.0269, Y 49.3989, Z -7.1667, A 0.000, B 0.000, C 0.000 }
gfCNCPoint5[12498] = {X 101.0176, Y 49.2586, Z -7.1667, A 0.000, B 0.000, C 0.000 }
gfCNCPoint5[12499] = {X 100.0676, Y 48.8899, Z -7.1667, A 0.000, B 0.000, C 0.000 }
gfCNCPoint5[12500] = {X 99.2280, Y 48.3125, Z -7.1667, A 0.000, B 0.000, C 0.000 }
gfCNCPoint5[12501] = {X 98.5436, Y 47.5575, Z -7.1667, A 0.000, B 0.000, C 0.000 }
gfCNCPoint5[12502] = {X 98.0514, Y 46.6653, Z -7.1667, A 0.000, B 0.000, C 0.000 }
gfCNCPoint5[12503] = {X 96.5892, Y 43.0894, Z -7.1667, A 0.000, B 0.000, C 0.000 }
gfCNCPoint5[12504] = {X 96.6993, Y 43.6444, Z -7.1667, A 0.000, B 0.000, C 0.000 }
gfCNCPoint5[12505] = {X 96.7385, Y 44.2089, Z -7.1667, A 0.000, B 0.000, C 0.000 }
gfCNCPoint5[12506] = {X 96.7383, Y 45.0423, Z -7.1667, A 0.000, B 0.000, C 0.000 }
gfCNCPoint5[12507] = {X 96.6200, Y 46.0144, Z -7.1667, A 0.000, B 0.000, C 0.000 }
gfCNCPoint5[12508] = {X 96.2896, Y 46.9363, Z -7.1667, A 0.000, B 0.000, C 0.000 }
gfCNCPoint5[12509] = {X 95.7635, Y 47.7622, Z -7.1667, A 0.000, B 0.000, C 0.000 }
gfCNCPoint5[12510] = {X 95.0677, Y 48.4513, Z -7.1667, A 0.000, B 0.000, C 0.000 }
gfCNCPoint5[12511] = {X 94.2367, Y 48.9695, Z -7.1667, A 0.000, B 0.000, C 0.000 }
gfCNCPoint5[12512] = {X 93.3117, Y 49.2910, Z -7.1667, A 0.000, B 0.000, C 0.000 }
gfCNCPoint5[12513] = {X 92.3385, Y 49.4000, Z -7.1667, A 0.000, B 0.000, C 0.000 }
gfCNCPoint5[12514] = {X 85.8951, Y 49.4000, Z -7.1667, A 0.000, B 0.000, C 0.000 }
gfCNCPoint5[12515] = {X 84.9160, Y 49.2897, Z -7.1667, A 0.000, B 0.000, C 0.000 }
gfCNCPoint5[12516] = {X 83.9860, Y 48.9643, Z -7.1667, A 0.000, B 0.000, C 0.000 }
gfCNCPoint5[12517] = {X 83.1517, Y 48.4401, Z -7.1667, A 0.000, B 0.000, C 0.000 }
gfCNCPoint5[12518] = {X 82.4550, Y 47.7433, Z -7.1667, A 0.000, B 0.000, C 0.000 }
gfCNCPoint5[12519] = {X 81.9308, Y 46.9091, Z -7.1667, A 0.000, B 0.000, C 0.000 }
gfCNCPoint5[12520] = {X 81.6054, Y 45.9791, Z -7.1667, A 0.000, B 0.000, C 0.000 }
gfCNCPoint5[12521] = {X 81.4951, Y 45.0000, Z -7.1667, A 0.000, B 0.000, C 0.000 }
gfCNCPoint5[12522] = {X 81.4951, Y 44.2068, Z -7.1667, A 0.000, B 0.000, C 0.000 }
gfCNCPoint5[12523] = {X 81.5997, Y 43.2694, Z -7.1667, A 0.000, B 0.000, C 0.000 }
gfCNCPoint5[12524] = {X 81.8993, Y 42.3750, Z -7.1667, A 0.000, B 0.000, C 0.000 }
gfCNCPoint5[12525] = {X 82.3806, Y 41.5637, Z -7.1667, A 0.000, B 0.000, C 0.000 }
gfCNCPoint5[12526] = {X 83.0219, Y 40.8720, Z -7.1667, A 0.000, B 0.000, C 0.000 }
gfCNCPoint5[12527] = {X 83.0217, Y 16.3102, Z -7.1667, A 0.000, B 0.000, C 0.000 }
gfCNCPoint5[12528] = {X 82.3774, Y 15.6212, Z -7.1667, A 0.000, B 0.000, C 0.000 }
gfCNCPoint5[12529] = {X 81.8949, Y 14.8106, Z -7.1667, A 0.000, B 0.000, C 0.000 }
gfCNCPoint5[12530] = {X 81.5962, Y 13.9158, Z -7.1667, A 0.000, B 0.000, C 0.000 }
gfCNCPoint5[12531] = {X 81.4951, Y 12.9780, Z -7.1667, A 0.000, B 0.000, C 0.000 }
gfCNCPoint5[12532] = {X 81.4951, Y 12.1868, Z -7.1667, A 0.000, B 0.000, C 0.000 }
gfCNCPoint5[12533] = {X 81.5776, Y 11.3388, Z -7.1667, A 0.000, B 0.000, C 0.000 }
gfCNCPoint5[12534] = {X 81.8220, Y 10.5225, Z -7.1667, A 0.000, B 0.000, C 0.000 }
gfCNCPoint5[12535] = {X 82.2191, Y 9.7687, Z -7.1667, A 0.000, B 0.000, C 0.000 }
gfCNCPoint5[12536] = {X 81.8181, Y 9.5049, Z -7.1667, A 0.000, B 0.000, C 0.000 }
gfCNCPoint5[12537] = {X 68.9232, Y 9.5049, Z -7.1667, A 0.000, B 0.000, C 0.000 }
gfCNCPoint5[12538] = {X 69.1905, Y 10.7207, Z -7.1667, A 0.000, B 0.000, C 0.000 }
gfCNCPoint5[12539] = {X 69.2995, Y 11.9609, Z -7.1667, A 0.000, B 0.000, C 0.000 }
gfCNCPoint5[12540] = {X 69.3015, Y 12.0738, Z -7.1667, A 0.000, B 0.000, C 0.000 }
gfCNCPoint5[12541] = {X 69.3021, Y 12.1868, Z -7.1667, A 0.000, B 0.000, C 0.000 }
gfCNCPoint5[12542] = {X 69.3017, Y 13.0687, Z -7.1667, A 0.000, B 0.000, C 0.000 }
gfCNCPoint5[12543] = {X 69.2128, Y 14.2899, Z -7.1667, A 0.000, B 0.000, C 0.000 }
gfCNCPoint5[12544] = {X 68.9705, Y 15.4901, Z -7.1667, A 0.000, B 0.000, C 0.000 }
gfCNCPoint5[12545] = {X 76.9197, Y 36.7543, Z -7.1667, A 0.000, B 0.000, C 0.000 }
gfCNCPoint5[12546] = {X 77.6315, Y 37.4065, Z -7.1667, A 0.000, B 0.000, C 0.000 }
gfCNCPoint5[12547] = {X 78.2748, Y 38.1263, Z -7.1667, A 0.000, B 0.000, C 0.000 }
gfCNCPoint5[12548] = {X 79.0226, Y 39.1913, Z -7.1667, A 0.000, B 0.000, C 0.000 }
gfCNCPoint5[12549] = {X 79.6208, Y 40.3470, Z -7.1667, A 0.000, B 0.000, C 0.000 }
gfCNCPoint5[12550] = {X 80.0585, Y 41.5724, Z -7.1667, A 0.000, B 0.000, C 0.000 }
gfCNCPoint5[12551] = {X 80.3280, Y 42.8455, Z -7.1667, A 0.000, B 0.000, C 0.000 }
gfCNCPoint5[12552] = {X 80.4242, Y 44.1432, Z -7.1667, A 0.000, B 0.000, C 0.000 }
gfCNCPoint5[12553] = {X 80.4245, Y 45.0000, Z -7.1667, A 0.000, B 0.000, C 0.000 }
gfCNCPoint5[12554] = {X 80.3511, Y 46.1898, Z -7.1667, A 0.000, B 0.000, C 0.000 }
gfCNCPoint5[12555] = {X 80.1320, Y 47.3615, Z -7.1667, A 0.000, B 0.000, C 0.000 }
gfCNCPoint5[12556] = {X 79.7706, Y 48.4974, Z -7.1667, A 0.000, B 0.000, C 0.000 }
gfCNCPoint5[12557] = {X 79.2722, Y 49.5803, Z -7.1667, A 0.000, B 0.000, C 0.000 }
gfCNCPoint5[12558] = {X 78.4688, Y 50.8341, Z -7.1667, A 0.000, B 0.000, C 0.000 }
gfCNCPoint5[12559] = {X 77.4826, Y 51.9498, Z -7.1667, A 0.000, B 0.000, C 0.000 }
gfCNCPoint5[12560] = {X 76.3369, Y 52.9011, Z -7.1667, A 0.000, B 0.000, C 0.000 }
gfCNCPoint5[12561] = {X 75.0589, Y 53.6653, Z -7.1667, A 0.000, B 0.000, C 0.000 }
gfCNCPoint5[12562] = {X 73.6787, Y 54.2246, Z -7.1667, A 0.000, B 0.000, C 0.000 }
gfCNCPoint5[12563] = {X 72.2292, Y 54.5655, Z -7.1667, A 0.000, B 0.000, C 0.000 }
gfCNCPoint5[12564] = {X 70.7445, Y 54.6800, Z -7.1667, A 0.000, B 0.000, C 0.000 }
gfCNCPoint5[12565] = {X 64.1851, Y 54.6800, Z -7.1667, A 0.000, B 0.000, C 0.000 }
gfCNCPoint5[12566] = {X 62.7229, Y 54.5689, Z -7.1667, A 0.000, B 0.000, C 0.000 }
gfCNCPoint5[12567] = {X 61.2943, Y 54.2383, Z -7.1667, A 0.000, B 0.000, C 0.000 }
gfCNCPoint5[12568] = {X 59.9320, Y 53.6956, Z -7.1667, A 0.000, B 0.000, C 0.000 }
gfCNCPoint5[12569] = {X 58.6673, Y 52.9534, Z -7.1667, A 0.000, B 0.000, C 0.000 }
gfCNCPoint5[12570] = {X 57.5293, Y 52.0286, Z -7.1667, A 0.000, B 0.000, C 0.000 }
gfCNCPoint5[12571] = {X 56.6337, Y 51.0563, Z -7.1667, A 0.000, B 0.000, C 0.000 }
gfCNCPoint5[12572] = {X 55.8790, Y 49.9710, Z -7.1667, A 0.000, B 0.000, C 0.000 }
gfCNCPoint5[12573] = {X 55.1243, Y 51.0563, Z -7.1667, A 0.000, B 0.000, C 0.000 }
gfCNCPoint5[12574] = {X 54.2288, Y 52.0286, Z -7.1667, A 0.000, B 0.000, C 0.000 }
gfCNCPoint5[12575] = {X 53.0907, Y 52.9534, Z -7.1667, A 0.000, B 0.000, C 0.000 }
gfCNCPoint5[12576] = {X 51.8261, Y 53.6956, Z -7.1667, A 0.000, B 0.000, C 0.000 }
gfCNCPoint5[12577] = {X 50.4638, Y 54.2383, Z -7.1667, A 0.000, B 0.000, C 0.000 }
gfCNCPoint5[12578] = {X 49.0351, Y 54.5689, Z -7.1667, A 0.000, B 0.000, C 0.000 }
gfCNCPoint5[12579] = {X 47.5729, Y 54.6800, Z -7.1667, A 0.000, B 0.000, C 0.000 }
gfCNCPoint5[12580] = {X 40.6393, Y 54.6800, Z -7.1667, A 0.000, B 0.000, C 0.000 }
gfCNCPoint5[12581] = {X 39.2448, Y 54.5790, Z -7.1667, A 0.000, B 0.000, C 0.000 }
gfCNCPoint5[12582] = {X 37.8793, Y 54.2782, Z -7.1667, A 0.000, B 0.000, C 0.000 }
gfCNCPoint5[12583] = {X 36.5715, Y 53.7838, Z -7.1667, A 0.000, B 0.000, C 0.000 }
gfCNCPoint5[12584] = {X 35.3485, Y 53.1062, Z -7.1667, A 0.000, B 0.000, C 0.000 }
gfCNCPoint5[12585] = {X 33.9155, Y 54.1348, Z -7.1667, A 0.000, B 0.000, C 0.000 }
gfCNCPoint5[12586] = {X 32.3645, Y 54.9751, Z -7.1667, A 0.000, B 0.000, C 0.000 }
gfCNCPoint5[12587] = {X 30.7203, Y 55.6139, Z -7.1667, A 0.000, B 0.000, C 0.000 }
gfCNCPoint5[12588] = {X 29.0088, Y 56.0411, Z -7.1667, A 0.000, B 0.000, C 0.000 }
gfCNCPoint5[12589] = {X 27.2572, Y 56.2498, Z -7.1667, A 0.000, B 0.000, C 0.000 }
gfCNCPoint5[12590] = {X 24.9790, Y 57.2346, Z -7.1667, A 0.000, B 0.000, C 0.000 }
gfCNCPoint5[12591] = {X 22.6425, Y 58.0720, Z -7.1667, A 0.000, B 0.000, C 0.000 }
gfCNCPoint5[12592] = {X 20.0815, Y 58.8002, Z -7.1667, A 0.000, B 0.000, C 0.000 }
gfCNCPoint5[12593] = {X 17.4693, Y 59.3160, Z -7.1667, A 0.000, B 0.000, C 0.000 }
gfCNCPoint5[12594] = {X 14.8237, Y 59.6157, Z -7.1667, A 0.000, B 0.000, C 0.000 }
gfCNCPoint5[12595] = {X 12.1624, Y 59.6974, Z -7.1667, A 0.000, B 0.000, C 0.000 }
gfCNCPoint5[12596] = {X 9.5033, Y 59.5606, Z -7.1667, A 0.000, B 0.000, C 0.000 }
gfCNCPoint5[12597] = {X 9.5033, Y 90.4951, Z -7.1667, A 0.000, B 0.000, C 0.000 }
gfCNCPoint5[12598] = {X 114.8626, Y 90.4951, Z -7.1667, A 0.000, B 0.000, C 0.000 }
gfCNCPoint5[12599] = {X 115.7469, Y 89.2983, Z -7.1667, A 0.000, B 0.000, C 0.000 }
gfCNCPoint5[12600] = {X 116.7716, Y 88.2192, Z -7.1667, A 0.000, B 0.000, C 0.000 }
gfCNCPoint5[12601] = {X 117.9212, Y 87.2744, Z -7.1667, A 0.000, B 0.000, C 0.000 }
gfCNCPoint5[12602] = {X 119.1783, Y 86.4780, Z -7.1667, A 0.000, B 0.000, C 0.000 }
gfCNCPoint5[12603] = {X 120.5237, Y 85.8423, Z -7.1667, A 0.000, B 0.000, C 0.000 }
gfCNCPoint5[12604] = {X 121.9371, Y 85.3768, Z -7.1667, A 0.000, B 0.000, C 0.000 }
gfCNCPoint5[12605] = {X 123.3970, Y 85.0886, Z -7.1667, A 0.000, B 0.000, C 0.000 }
gfCNCPoint5[12606] = {X 123.5296, Y 84.9453, Z -7.1667, A 0.000, B 0.000, C 0.000 }
gfCNCPoint5[12607] = {X 123.6609, Y 84.8009, Z -7.1667, A 0.000, B 0.000, C 0.000 }
gfCNCPoint5[12608] = {X 147.2181, Y 58.9335, Z -7.1667, A 0.000, B 0.000, C 0.000 }
gfCNCPoint5[12609] = {X 147.2180, Y 58.0000, Z -7.1667, A 0.000, B 0.000, C 0.000 }
gfCNCPoint5[12610] = {X 147.2987, Y 56.6058, Z -7.1667, A 0.000, B 0.000, C 0.000 }
gfCNCPoint5[12611] = {X 147.5398, Y 55.2303, Z -7.1667, A 0.000, B 0.000, C 0.000 }
gfCNCPoint5[12612] = {X 148.0022, Y 53.7185, Z -7.1667, A 0.000, B 0.000, C 0.000 }
gfCNCPoint5[12613] = {X 148.6580, Y 52.2800, Z -7.1667, A 0.000, B 0.000, C 0.000 }
gfCNCPoint5[12614] = {X 143.0396, Y 52.2800, Z -7.1667, A 0.000, B 0.000, C 0.000 }
gfCNCPoint5[12615] = {X 141.7807, Y 52.1703, Z -7.1667, A 0.000, B 0.000, C 0.000 }
gfCNCPoint5[12616] = {X 140.5597, Y 51.8446, Z -7.1667, A 0.000, B 0.000, C 0.000 }
gfCNCPoint5[12617] = {X 139.4134, Y 51.3126, Z -7.1667, A 0.000, B 0.000, C 0.000 }
gfCNCPoint5[12618] = {X 138.3764, Y 50.5904, Z -7.1667, A 0.000, B 0.000, C 0.000 }
gfCNCPoint5[12619] = {X 137.4799, Y 49.6998, Z -7.1667, A 0.000, B 0.000, C 0.000 }
gfCNCPoint5[12620] = {X 136.7509, Y 48.6675, Z -7.1667, A 0.000, B 0.000, C 0.000 }
gfCNCPoint5[12621] = {X 136.2114, Y 47.5248, Z -7.1667, A 0.000, B 0.000, C 0.000 }
gfCNCPoint5[12622] = {X 135.8777, Y 46.3059, Z -7.1667, A 0.000, B 0.000, C 0.000 }
gfCNCPoint5[12623] = {X 135.7598, Y 45.0477, Z -7.1667, A 0.000, B 0.000, C 0.000 }
gfCNCPoint5[12624] = {X 135.7601, Y 44.1248, Z -7.1667, A 0.000, B 0.000, C 0.000 }
gfCNCPoint5[12625] = {X 135.8408, Y 43.1249, Z -7.1667, A 0.000, B 0.000, C 0.000 }
gfCNCPoint5[12626] = {X 136.0581, Y 42.1457, Z -7.1667, A 0.000, B 0.000, C 0.000 }
gfCNCPoint5[12627] = {X 138.3597, Y 42.8258, Z -7.1667, A 0.000, B 0.000, C 0.000 }
gfCNCPoint5[12628] = {X 138.6721, Y 42.0319, Z -7.1667, A 0.000, B 0.000, C 0.000 }
gfCNCPoint5[12629] = {X 139.1179, Y 41.3046, Z -7.1667, A 0.000, B 0.000, C 0.000 }
gfCNCPoint5[12630] = {X 139.6836, Y 40.6660, Z -7.1667, A 0.000, B 0.000, C 0.000 }
gfCNCPoint5[12631] = {X 139.6836, Y 20.4382, Z -7.1667, A 0.000, B 0.000, C 0.000 }
gfCNCPoint5[12632] = {X 137.7096, Y 20.4379, Z -7.1667, A 0.000, B 0.000, C 0.000 }
gfCNCPoint5[12633] = {X 136.9995, Y 21.1826, Z -7.1667, A 0.000, B 0.000, C 0.000 }
gfCNCPoint5[12634] = {X 136.1491, Y 21.7619, Z -7.1667, A 0.000, B 0.000, C 0.000 }
gfCNCPoint5[12635] = {X 135.4282, Y 22.0767, Z -7.1667, A 0.000, B 0.000, C 0.000 }
gfCNCPoint5[12636] = {X 134.6660, Y 22.2715, Z -7.1667, A 0.000, B 0.000, C 0.000 }
gfCNCPoint5[12637] = {X 133.8824, Y 22.3414, Z -7.1667, A 0.000, B 0.000, C 0.000 }
gfCNCPoint5[12638] = {X 133.2006, Y 22.3415, Z -7.1667, A 0.000, B 0.000, C 0.000 }
gfCNCPoint5[12639] = {X 132.2486, Y 22.2478, Z -7.1667, A 0.000, B 0.000, C 0.000 }
gfCNCPoint5[12640] = {X 131.3331, Y 21.9701, Z -7.1667, A 0.000, B 0.000, C 0.000 }
gfCNCPoint5[12641] = {X 130.4895, Y 21.5191, Z -7.1667, A 0.000, B 0.000, C 0.000 }
gfCNCPoint5[12642] = {X 129.7500, Y 20.9122, Z -7.1667, A 0.000, B 0.000, C 0.000 }
gfCNCPoint5[12643] = {X 129.1431, Y 20.1727, Z -7.1667, A 0.000, B 0.000, C 0.000 }
gfCNCPoint5[12644] = {X 128.6921, Y 19.3290, Z -7.1667, A 0.000, B 0.000, C 0.000 }
gfCNCPoint5[12645] = {X 128.4144, Y 18.4136, Z -7.1667, A 0.000, B 0.000, C 0.000 }
gfCNCPoint5[12646] = {X 128.3206, Y 17.4615, Z -7.1667, A 0.000, B 0.000, C 0.000 }
gfCNCPoint5[12647] = {X 128.3206, Y 10.4835, Z -7.1667, A 0.000, B 0.000, C 0.000 }
gfCNCPoint5[12648] = {X 128.3317, Y 10.1548, Z -7.1667, A 0.000, B 0.000, C 0.000 }
gfCNCPoint5[12649] = {X 128.3649, Y 9.8275, Z -7.1667, A 0.000, B 0.000, C 0.000 }
gfCNCPoint5[12650] = {X 128.6079, Y 8.8340, Z -7.1667, A 0.000, B 0.000, C 0.000 }
gfCNCPoint5[12651] = {X 129.0525, Y 7.9130, Z -7.1667, A 0.000, B 0.000, C 0.000 }
gfCNCPoint5[12652] = {X 129.6794, Y 7.1049, Z -7.1667, A 0.000, B 0.000, C 0.000 }
gfCNCPoint5[12653] = {X 130.0258, Y 7.4372, Z -7.1667, A 0.000, B 0.000, C 0.000 }
gfCNCPoint5[12654] = {X 130.6997, Y 6.8634, Z -7.1667, A 0.000, B 0.000, C 0.000 }
gfCNCPoint5[12655] = {X 131.4749, Y 6.4361, Z -7.1667, A 0.000, B 0.000, C 0.000 }
gfCNCPoint5[12656] = {X 132.3200, Y 6.1726, Z -7.1667, A 0.000, B 0.000, C 0.000 }
gfCNCPoint5[12657] = {X 133.2007, Y 6.0835, Z -7.1667, A 0.000, B 0.000, C 0.000 }
gfCNCPoint5[12658] = {X 133.8874, Y 6.0837, Z -7.1667, A 0.000, B 0.000, C 0.000 }
gfCNCPoint5[12659] = {X 134.7186, Y 6.1717, Z -7.1667, A 0.000, B 0.000, C 0.000 }
gfCNCPoint5[12660] = {X 135.5182, Y 6.4152, Z -7.1667, A 0.000, B 0.000, C 0.000 }
gfCNCPoint5[12661] = {X 136.2572, Y 6.8055, Z -7.1667, A 0.000, B 0.000, C 0.000 }
gfCNCPoint5[12662] = {X 136.9092, Y 7.3285, Z -7.1667, A 0.000, B 0.000, C 0.000 }
gfCNCPoint5[12663] = {X 137.4505, Y 7.9654, Z -7.1667, A 0.000, B 0.000, C 0.000 }
gfCNCPoint5[12664] = {X 155.0722, Y 7.9654, Z -7.1667, A 0.000, B 0.000, C 0.000 }
gfCNCPoint5[12665] = {X 155.6200, Y 7.3222, Z -7.1667, A 0.000, B 0.000, C 0.000 }
gfCNCPoint5[12666] = {X 156.2806, Y 6.7956, Z -7.1667, A 0.000, B 0.000, C 0.000 }
gfCNCPoint5[12667] = {X 157.0297, Y 6.4049, Z -7.1667, A 0.000, B 0.000, C 0.000 }
gfCNCPoint5[12668] = {X 157.8396, Y 6.1646, Z -7.1667, A 0.000, B 0.000, C 0.000 }
gfCNCPoint5[12669] = {X 158.6805, Y 6.0835, Z -7.1667, A 0.000, B 0.000, C 0.000 }
gfCNCPoint5[12670] = {X 159.3791, Y 6.0839, Z -7.1667, A 0.000, B 0.000, C 0.000 }
gfCNCPoint5[12671] = {X 160.3488, Y 6.2050, Z -7.1667, A 0.000, B 0.000, C 0.000 }
gfCNCPoint5[12672] = {X 161.2678, Y 6.5371, Z -7.1667, A 0.000, B 0.000, C 0.000 }
gfCNCPoint5[12673] = {X 162.0908, Y 7.0639, Z -7.1667, A 0.000, B 0.000, C 0.000 }
gfCNCPoint5[12674] = {X 162.7773, Y 7.7593, Z -7.1667, A 0.000, B 0.000, C 0.000 }
gfCNCPoint5[12675] = {X 163.2934, Y 8.5891, Z -7.1667, A 0.000, B 0.000, C 0.000 }
gfCNCPoint5[12676] = {X 163.6136, Y 9.5124, Z -7.1667, A 0.000, B 0.000, C 0.000 }
gfCNCPoint5[12677] = {X 163.7221, Y 10.4835, Z -7.1667, A 0.000, B 0.000, C 0.000 }
gfCNCPoint5[12678] = {X 163.7221, Y 17.4615, Z -7.1667, A 0.000, B 0.000, C 0.000 }
gfCNCPoint5[12679] = {X 163.6118, Y 18.4406, Z -7.1667, A 0.000, B 0.000, C 0.000 }
gfCNCPoint5[12680] = {X 163.2863, Y 19.3706, Z -7.1667, A 0.000, B 0.000, C 0.000 }
gfCNCPoint5[12681] = {X 162.7621, Y 20.2049, Z -7.1667, A 0.000, B 0.000, C 0.000 }
gfCNCPoint5[12682] = {X 162.0654, Y 20.9016, Z -7.1667, A 0.000, B 0.000, C 0.000 }
gfCNCPoint5[12683] = {X 161.2312, Y 21.4258, Z -7.1667, A 0.000, B 0.000, C 0.000 }
gfCNCPoint5[12684] = {X 160.3012, Y 21.7512, Z -7.1667, A 0.000, B 0.000, C 0.000 }
gfCNCPoint5[12685] = {X 159.3221, Y 21.8615, Z -7.1667, A 0.000, B 0.000, C 0.000 }
gfCNCPoint5[12686] = {X 158.6791, Y 21.8615, Z -7.1667, A 0.000, B 0.000, C 0.000 }
gfCNCPoint5[12687] = {X 157.8336, Y 21.7771, Z -7.1667, A 0.000, B 0.000, C 0.000 }
gfCNCPoint5[12688] = {X 157.0198, Y 21.5329, Z -7.1667, A 0.000, B 0.000, C 0.000 }
gfCNCPoint5[12689] = {X 156.2675, Y 21.1377, Z -7.1667, A 0.000, B 0.000, C 0.000 }
gfCNCPoint5[12690] = {X 155.6046, Y 20.6062, Z -7.1667, A 0.000, B 0.000, C 0.000 }
gfCNCPoint5[12691] = {X 155.0553, Y 19.9579, Z -7.1667, A 0.000, B 0.000, C 0.000 }
gfCNCPoint5[12692] = {X 152.3572, Y 19.9588, Z -7.1667, A 0.000, B 0.000, C 0.000 }
gfCNCPoint5[12693] = {X 152.3561, Y 40.8428, Z -7.1667, A 0.000, B 0.000, C 0.000 }
gfCNCPoint5[12694] = {X 152.8071, Y 41.3291, Z -7.1667, A 0.000, B 0.000, C 0.000 }
gfCNCPoint5[12695] = {X 152.9010, Y 41.4409, Z -7.1667, A 0.000, B 0.000, C 0.000 }
gfCNCPoint5[12696] = {X 153.4354, Y 42.2812, Z -7.1667, A 0.000, B 0.000, C 0.000 }
gfCNCPoint5[12697] = {X 153.7684, Y 43.2197, Z -7.1667, A 0.000, B 0.000, C 0.000 }
gfCNCPoint5[12698] = {X 153.8831, Y 44.2088, Z -7.1667, A 0.000, B 0.000, C 0.000 }
gfCNCPoint5[12699] = {X 153.8829, Y 45.0423, Z -7.1667, A 0.000, B 0.000, C 0.000 }
gfCNCPoint5[12700] = {X 153.7646, Y 46.0144, Z -7.1667, A 0.000, B 0.000, C 0.000 }
gfCNCPoint5[12701] = {X 153.4342, Y 46.9363, Z -7.1667, A 0.000, B 0.000, C 0.000 }
gfCNCPoint5[12702] = {X 152.9080, Y 47.7622, Z -7.1667, A 0.000, B 0.000, C 0.000 }
gfCNCPoint5[12703] = {X 152.2123, Y 48.4513, Z -7.1667, A 0.000, B 0.000, C 0.000 }
gfCNCPoint5[12704] = {X 151.3813, Y 48.9695, Z -7.1667, A 0.000, B 0.000, C 0.000 }
gfCNCPoint5[12705] = {X 150.4563, Y 49.2910, Z -7.1667, A 0.000, B 0.000, C 0.000 }
gfCNCPoint5[12706] = {X 149.4831, Y 49.4000, Z -7.1667, A 0.000, B 0.000, C 0.000 }
gfCNCPoint5[12707] = {X 143.0396, Y 49.4000, Z -7.1667, A 0.000, B 0.000, C 0.000 }
gfCNCPoint5[12708] = {X 142.0605, Y 49.2897, Z -7.1667, A 0.000, B 0.000, C 0.000 }
gfCNCPoint5[12709] = {X 141.1305, Y 48.9643, Z -7.1667, A 0.000, B 0.000, C 0.000 }
gfCNCPoint5[12710] = {X 140.2963, Y 48.4400, Z -7.1667, A 0.000, B 0.000, C 0.000 }
gfCNCPoint5[12711] = {X 139.5996, Y 47.7433, Z -7.1667, A 0.000, B 0.000, C 0.000 }
gfCNCPoint5[12712] = {X 139.0754, Y 46.9091, Z -7.1667, A 0.000, B 0.000, C 0.000 }
gfCNCPoint5[12713] = {X 138.7499, Y 45.9791, Z -7.1667, A 0.000, B 0.000, C 0.000 }
gfCNCPoint5[12714] = {X 138.6396, Y 45.0000, Z -7.1667, A 0.000, B 0.000, C 0.000 }
gfCNCPoint5[12715] = {X 138.6400, Y 44.1483, Z -7.1667, A 0.000, B 0.000, C 0.000 }
gfCNCPoint5[12716] = {X 138.7505, Y 43.2275, Z -7.1667, A 0.000, B 0.000, C 0.000 }
gfCNCPoint5[12717] = {X 139.0514, Y 42.3503, Z -7.1667, A 0.000, B 0.000, C 0.000 }
gfCNCPoint5[12718] = {X 139.5295, Y 41.5556, Z -7.1667, A 0.000, B 0.000, C 0.000 }
gfCNCPoint5[12719] = {X 140.1636, Y 40.8789, Z -7.1667, A 0.000, B 0.000, C 0.000 }
gfCNCPoint5[12720] = {X 140.1636, Y 19.9582, Z -7.1667, A 0.000, B 0.000, C 0.000 }
gfCNCPoint5[12721] = {X 137.4656, Y 19.9579, Z -7.1667, A 0.000, B 0.000, C 0.000 }
gfCNCPoint5[12722] = {X 136.9179, Y 20.6081, Z -7.1667, A 0.000, B 0.000, C 0.000 }
gfCNCPoint5[12723] = {X 136.2554, Y 21.1408, Z -7.1667, A 0.000, B 0.000, C 0.000 }
gfCNCPoint5[12724] = {X 135.5029, Y 21.5362, Z -7.1667, A 0.000, B 0.000, C 0.000 }
gfCNCPoint5[12725] = {X 134.6883, Y 21.7794, Z -7.1667, A 0.000, B 0.000, C 0.000 }
gfCNCPoint5[12726] = {X 133.8422, Y 21.8615, Z -7.1667, A 0.000, B 0.000, C 0.000 }
gfCNCPoint5[12727] = {X 133.2006, Y 21.8615, Z -7.1667, A 0.000, B 0.000, C 0.000 }
gfCNCPoint5[12728] = {X 132.2215, Y 21.7512, Z -7.1667, A 0.000, B 0.000, C 0.000 }
gfCNCPoint5[12729] = {X 131.2916, Y 21.4258, Z -7.1667, A 0.000, B 0.000, C 0.000 }
gfCNCPoint5[12730] = {X 130.4573, Y 20.9016, Z -7.1667, A 0.000, B 0.000, C 0.000 }
gfCNCPoint5[12731] = {X 129.7606, Y 20.2049, Z -7.1667, A 0.000, B 0.000, C 0.000 }
gfCNCPoint5[12732] = {X 129.2364, Y 19.3706, Z -7.1667, A 0.000, B 0.000, C 0.000 }
gfCNCPoint5[12733] = {X 128.9110, Y 18.4406, Z -7.1667, A 0.000, B 0.000, C 0.000 }
gfCNCPoint5[12734] = {X 128.8006, Y 17.4615, Z -7.1667, A 0.000, B 0.000, C 0.000 }
gfCNCPoint5[12735] = {X 128.8006, Y 10.4835, Z -7.1667, A 0.000, B 0.000, C 0.000 }
gfCNCPoint5[12736] = {X 128.8808, Y 9.6474, Z -7.1667, A 0.000, B 0.000, C 0.000 }
gfCNCPoint5[12737] = {X 129.1184, Y 8.8418, Z -7.1667, A 0.000, B 0.000, C 0.000 }
gfCNCPoint5[12738] = {X 129.5047, Y 8.0960, Z -7.1667, A 0.000, B 0.000, C 0.000 }
gfCNCPoint5[12739] = {X 130.0258, Y 7.4372, Z -7.1667, A 0.000, B 0.000, C 0.000 }
gfCNCPoint5[12740] = {X 129.6794, Y 7.1049, Z -7.1667, A 0.000, B 0.000, C 0.000 }
gfCNCPoint5[12741] = {X 102.4337, Y 7.1049, Z -7.1667, A 0.000, B 0.000, C 0.000 }
gfCNCPoint5[12742] = {X 102.4337, Y 11.9049, Z -7.1667, A 0.000, B 0.000, C 0.000 }
gfCNCPoint5[12743] = {X 101.3242, Y 11.9049, Z -7.1667, A 0.000, B 0.000, C 0.000 }
gfCNCPoint5[12744] = {X 101.3283, Y 12.0458, Z -7.1667, A 0.000, B 0.000, C 0.000 }
gfCNCPoint5[12745] = {X 101.3297, Y 12.1868, Z -7.1667, A 0.000, B 0.000, C 0.000 }
gfCNCPoint5[12746] = {X 101.3293, Y 13.0462, Z -7.1667, A 0.000, B 0.000, C 0.000 }
gfCNCPoint5[12747] = {X 101.2278, Y 14.1915, Z -7.1667, A 0.000, B 0.000, C 0.000 }
gfCNCPoint5[12748] = {X 100.9472, Y 15.3065, Z -7.1667, A 0.000, B 0.000, C 0.000 }
gfCNCPoint5[12749] = {X 101.8689, Y 17.5912, Z -7.1667, A 0.000, B 0.000, C 0.000 }
gfCNCPoint5[12750] = {X 102.3680, Y 16.3467, Z -7.1667, A 0.000, B 0.000, C 0.000 }
gfCNCPoint5[12751] = {X 102.7994, Y 15.2726, Z -7.1667, A 0.000, B 0.000, C 0.000 }
gfCNCPoint5[12752] = {X 102.5271, Y 14.1735, Z -7.1667, A 0.000, B 0.000, C 0.000 }
gfCNCPoint5[12753] = {X 102.4286, Y 13.0454, Z -7.1667, A 0.000, B 0.000, C 0.000 }
gfCNCPoint5[12754] = {X 102.4283, Y 12.1868, Z -7.1667, A 0.000, B 0.000, C 0.000 }
gfCNCPoint5[12755] = {X 102.4296, Y 12.0458, Z -7.1667, A 0.000, B 0.000, C 0.000 }
gfCNCPoint5[12756] = {X 102.4337, Y 11.9049, Z -7.1667, A 0.000, B 0.000, C 0.000 }
gfCNCPoint5[12757] = {X 102.4337, Y 9.5049, Z -7.1667, A 0.000, B 0.000, C 0.000 }
gfCNCPoint5[12758] = {X 98.1266, Y 9.5049, Z -7.1667, A 0.000, B 0.000, C 0.000 }
gfCNCPoint5[12759] = {X 98.5429, Y 10.2828, Z -7.1667, A 0.000, B 0.000, C 0.000 }
gfCNCPoint5[12760] = {X 98.8123, Y 11.1229, Z -7.1667, A 0.000, B 0.000, C 0.000 }
gfCNCPoint5[12761] = {X 98.9260, Y 11.9978, Z -7.1667, A 0.000, B 0.000, C 0.000 }
gfCNCPoint5[12762] = {X 98.9288, Y 12.0923, Z -7.1667, A 0.000, B 0.000, C 0.000 }
gfCNCPoint5[12763] = {X 98.9297, Y 12.1868, Z -7.1667, A 0.000, B 0.000, C 0.000 }
gfCNCPoint5[12764] = {X 98.9294, Y 13.0237, Z -7.1667, A 0.000, B 0.000, C 0.000 }
gfCNCPoint5[12765] = {X 98.8591, Y 13.8052, Z -7.1667, A 0.000, B 0.000, C 0.000 }
gfCNCPoint5[12766] = {X 98.6643, Y 14.5652, Z -7.1667, A 0.000, B 0.000, C 0.000 }
gfCNCPoint5[12767] = {X 98.3503, Y 15.2843, Z -7.1667, A 0.000, B 0.000, C 0.000 }
gfCNCPoint5[12768] = {X 101.8754, Y 24.0228, Z -7.1667, A 0.000, B 0.000, C 0.000 }
gfCNCPoint5[12769] = {X 104.5953, Y 17.2406, Z -7.1667, A 0.000, B 0.000, C 0.000 }
gfCNCPoint5[12770] = {X 105.3925, Y 15.2558, Z -7.1667, A 0.000, B 0.000, C 0.000 }
gfCNCPoint5[12771] = {X 105.0866, Y 14.5447, Z -7.1667, A 0.000, B 0.000, C 0.000 }
gfCNCPoint5[12772] = {X 104.8970, Y 13.7941, Z -7.1667, A 0.000, B 0.000, C 0.000 }
gfCNCPoint5[12773] = {X 104.8285, Y 13.0231, Z -7.1667, A 0.000, B 0.000, C 0.000 }
gfCNCPoint5[12774] = {X 104.8283, Y 12.1868, Z -7.1667, A 0.000, B 0.000, C 0.000 }
gfCNCPoint5[12775] = {X 104.8292, Y 12.0923, Z -7.1667, A 0.000, B 0.000, C 0.000 }
gfCNCPoint5[12776] = {X 104.8319, Y 11.9978, Z -7.1667, A 0.000, B 0.000, C 0.000 }
gfCNCPoint5[12777] = {X 104.9457, Y 11.1229, Z -7.1667, A 0.000, B 0.000, C 0.000 }
gfCNCPoint5[12778] = {X 105.2151, Y 10.2828, Z -7.1667, A 0.000, B 0.000, C 0.000 }
gfCNCPoint5[12779] = {X 105.6313, Y 9.5049, Z -7.1667, A 0.000, B 0.000, C 0.000 }
gfCNCPoint5[12780] = {X 102.4337, Y 9.5049, Z -7.1667, A 0.000, B 0.000, C 0.000 }
gfCNCPoint5[12781] = {X 102.4337, Y 7.1049, Z -7.1667, A 0.000, B 0.000, C 0.000 }
gfCNCPoint5[12782] = {X 64.8348, Y 7.1049, Z -7.1667, A 0.000, B 0.000, C 0.000 }
gfCNCPoint5[12783] = {X 65.5945, Y 8.0240, Z -7.1667, A 0.000, B 0.000, C 0.000 }
gfCNCPoint5[12784] = {X 66.1940, Y 9.0549, Z -7.1667, A 0.000, B 0.000, C 0.000 }
gfCNCPoint5[12785] = {X 66.6171, Y 10.1698, Z -7.1667, A 0.000, B 0.000, C 0.000 }
gfCNCPoint5[12786] = {X 66.8305, Y 11.1683, Z -7.1667, A 0.000, B 0.000, C 0.000 }
gfCNCPoint5[12787] = {X 66.9021, Y 12.1868, Z -7.1667, A 0.000, B 0.000, C 0.000 }
gfCNCPoint5[12788] = {X 66.9018, Y 13.0462, Z -7.1667, A 0.000, B 0.000, C 0.000 }
gfCNCPoint5[12789] = {X 66.7773, Y 14.3202, Z -7.1667, A 0.000, B 0.000, C 0.000 }
gfCNCPoint5[12790] = {X 66.4316, Y 15.5527, Z -7.1667, A 0.000, B 0.000, C 0.000 }
gfCNCPoint5[12791] = {X 74.9130, Y 38.2404, Z -7.1667, A 0.000, B 0.000, C 0.000 }
gfCNCPoint5[12792] = {X 75.8049, Y 38.9752, Z -7.1667, A 0.000, B 0.000, C 0.000 }
gfCNCPoint5[12793] = {X 76.5693, Y 39.8419, Z -7.1667, A 0.000, B 0.000, C 0.000 }
gfCNCPoint5[12794] = {X 77.1869, Y 40.8186, Z -7.1667, A 0.000, B 0.000, C 0.000 }
gfCNCPoint5[12795] = {X 77.6422, Y 41.8807, Z -7.1667, A 0.000, B 0.000, C 0.000 }
gfCNCPoint5[12796] = {X 77.9237, Y 43.0015, Z -7.1667, A 0.000, B 0.000, C 0.000 }
gfCNCPoint5[12797] = {X 78.0243, Y 44.1527, Z -7.1667, A 0.000, B 0.000, C 0.000 }
gfCNCPoint5[12798] = {X 78.0245, Y 45.0000, Z -7.1667, A 0.000, B 0.000, C 0.000 }
gfCNCPoint5[12799] = {X 77.9139, Y 46.2642, Z -7.1667, A 0.000, B 0.000, C 0.000 }
gfCNCPoint5[12800] = {X 77.5854, Y 47.4899, Z -7.1667, A 0.000, B 0.000, C 0.000 }
gfCNCPoint5[12801] = {X 77.0491, Y 48.6400, Z -7.1667, A 0.000, B 0.000, C 0.000 }
gfCNCPoint5[12802] = {X 76.3213, Y 49.6795, Z -7.1667, A 0.000, B 0.000, C 0.000 }
gfCNCPoint5[12803] = {X 75.4240, Y 50.5768, Z -7.1667, A 0.000, B 0.000, C 0.000 }
gfCNCPoint5[12804] = {X 74.3845, Y 51.3047, Z -7.1667, A 0.000, B 0.000, C 0.000 }
gfCNCPoint5[12805] = {X 73.2344, Y 51.8410, Z -7.1667, A 0.000, B 0.000, C 0.000 }
gfCNCPoint5[12806] = {X 72.0086, Y 52.1694, Z -7.1667, A 0.000, B 0.000, C 0.000 }
gfCNCPoint5[12807] = {X 70.7445, Y 52.2800, Z -7.1667, A 0.000, B 0.000, C 0.000 }
gfCNCPoint5[12808] = {X 64.1851, Y 52.2800, Z -7.1667, A 0.000, B 0.000, C 0.000 }
gfCNCPoint5[12809] = {X 62.9397, Y 52.1727, Z -7.1667, A 0.000, B 0.000, C 0.000 }
gfCNCPoint5[12810] = {X 61.7311, Y 51.8539, Z -7.1667, A 0.000, B 0.000, C 0.000 }
gfCNCPoint5[12811] = {X 60.5947, Y 51.3330, Z -7.1667, A 0.000, B 0.000, C 0.000 }
gfCNCPoint5[12812] = {X 59.5643, Y 50.6255, Z -7.1667, A 0.000, B 0.000, C 0.000 }
gfCNCPoint5[12813] = {X 58.6700, Y 49.7521, Z -7.1667, A 0.000, B 0.000, C 0.000 }
gfCNCPoint5[12814] = {X 57.9384, Y 48.7385, Z -7.1667, A 0.000, B 0.000, C 0.000 }
gfCNCPoint5[12815] = {X 57.3706, Y 47.5614, Z -7.1667, A 0.000, B 0.000, C 0.000 }
gfCNCPoint5[12816] = {X 57.0224, Y 46.3017, Z -7.1667, A 0.000, B 0.000, C 0.000 }
gfCNCPoint5[12817] = {X 56.9051, Y 45.0000, Z -7.1667, A 0.000, B 0.000, C 0.000 }
gfCNCPoint5[12818] = {X 56.9051, Y 44.2048, Z -7.1667, A 0.000, B 0.000, C 0.000 }
gfCNCPoint5[12819] = {X 56.9286, Y 43.6251, Z -7.1667, A 0.000, B 0.000, C 0.000 }
gfCNCPoint5[12820] = {X 56.9981, Y 43.0492, Z -7.1667, A 0.000, B 0.000, C 0.000 }
gfCNCPoint5[12821] = {X 54.7600, Y 43.0492, Z -7.1667, A 0.000, B 0.000, C 0.000 }
gfCNCPoint5[12822] = {X 54.8275, Y 43.6012, Z -7.1667, A 0.000, B 0.000, C 0.000 }
gfCNCPoint5[12823] = {X 54.8528, Y 44.1567, Z -7.1667, A 0.000, B 0.000, C 0.000 }
gfCNCPoint5[12824] = {X 54.8529, Y 45.0000, Z -7.1667, A 0.000, B 0.000, C 0.000 }
gfCNCPoint5[12825] = {X 54.7356, Y 46.3017, Z -7.1667, A 0.000, B 0.000, C 0.000 }
gfCNCPoint5[12826] = {X 54.3875, Y 47.5614, Z -7.1667, A 0.000, B 0.000, C 0.000 }
gfCNCPoint5[12827] = {X 53.8197, Y 48.7385, Z -7.1667, A 0.000, B 0.000, C 0.000 }
gfCNCPoint5[12828] = {X 53.0880, Y 49.7521, Z -7.1667, A 0.000, B 0.000, C 0.000 }
gfCNCPoint5[12829] = {X 52.1938, Y 50.6255, Z -7.1667, A 0.000, B 0.000, C 0.000 }
gfCNCPoint5[12830] = {X 51.1633, Y 51.3330, Z -7.1667, A 0.000, B 0.000, C 0.000 }
gfCNCPoint5[12831] = {X 50.0270, Y 51.8539, Z -7.1667, A 0.000, B 0.000, C 0.000 }
gfCNCPoint5[12832] = {X 48.8183, Y 52.1727, Z -7.1667, A 0.000, B 0.000, C 0.000 }
gfCNCPoint5[12833] = {X 47.5729, Y 52.2800, Z -7.1667, A 0.000, B 0.000, C 0.000 }
gfCNCPoint5[12834] = {X 40.6393, Y 52.2800, Z -7.1667, A 0.000, B 0.000, C 0.000 }
gfCNCPoint5[12835] = {X 39.4476, Y 52.1818, Z -7.1667, A 0.000, B 0.000, C 0.000 }
gfCNCPoint5[12836] = {X 38.2881, Y 51.8899, Z -7.1667, A 0.000, B 0.000, C 0.000 }
gfCNCPoint5[12837] = {X 37.1919, Y 51.4120, Z -7.1667, A 0.000, B 0.000, C 0.000 }
gfCNCPoint5[12838] = {X 36.1888, Y 50.7612, Z -7.1667, A 0.000, B 0.000, C 0.000 }
gfCNCPoint5[12839] = {X 35.3058, Y 49.9550, Z -7.1667, A 0.000, B 0.000, C 0.000 }
gfCNCPoint5[12840] = {X 34.8234, Y 50.4196, Z -7.1667, A 0.000, B 0.000, C 0.000 }
gfCNCPoint5[12841] = {X 34.3150, Y 50.8555, Z -7.1667, A 0.000, B 0.000, C 0.000 }
gfCNCPoint5[12842] = {X 33.7800, Y 51.2881, Z -7.1667, A 0.000, B 0.000, C 0.000 }
gfCNCPoint5[12843] = {X 32.5213, Y 52.1749, Z -7.1667, A 0.000, B 0.000, C 0.000 }
gfCNCPoint5[12844] = {X 31.1563, Y 52.8873, Z -7.1667, A 0.000, B 0.000, C 0.000 }
gfCNCPoint5[12845] = {X 29.7090, Y 53.4129, Z -7.1667, A 0.000, B 0.000, C 0.000 }
gfCNCPoint5[12846] = {X 28.2049, Y 53.7423, Z -7.1667, A 0.000, B 0.000, C 0.000 }
gfCNCPoint5[12847] = {X 26.6705, Y 53.8699, Z -7.1667, A 0.000, B 0.000, C 0.000 }
gfCNCPoint5[12848] = {X 24.3184, Y 54.9142, Z -7.1667, A 0.000, B 0.000, C 0.000 }
gfCNCPoint5[12849] = {X 21.8986, Y 55.7903, Z -7.1667, A 0.000, B 0.000, C 0.000 }
gfCNCPoint5[12850] = {X 19.5258, Y 56.4655, Z -7.1667, A 0.000, B 0.000, C 0.000 }
gfCNCPoint5[12851] = {X 17.1056, Y 56.9437, Z -7.1667, A 0.000, B 0.000, C 0.000 }
gfCNCPoint5[12852] = {X 14.6544, Y 57.2217, Z -7.1667, A 0.000, B 0.000, C 0.000 }
gfCNCPoint5[12853] = {X 12.1886, Y 57.2976, Z -7.1667, A 0.000, B 0.000, C 0.000 }
gfCNCPoint5[12854] = {X 9.7249, Y 57.1709, Z -7.1667, A 0.000, B 0.000, C 0.000 }
gfCNCPoint5[12855] = {X 8.4102, Y 57.0197, Z -7.1667, A 0.000, B 0.000, C 0.000 }
gfCNCPoint5[12856] = {X 7.1033, Y 56.8107, Z -7.1667, A 0.000, B 0.000, C 0.000 }
gfCNCPoint5[12857] = {X 7.1033, Y 92.8951, Z -7.1667, A 0.000, B 0.000, C 0.000 }
gfCNCPoint5[12858] = {X 116.2646, Y 92.8951, Z -7.1667, A 0.000, B 0.000, C 0.000 }
gfCNCPoint5[12859] = {X 116.9733, Y 91.6540, Z -7.1667, A 0.000, B 0.000, C 0.000 }
gfCNCPoint5[12860] = {X 117.8570, Y 90.5308, Z -7.1667, A 0.000, B 0.000, C 0.000 }
gfCNCPoint5[12861] = {X 118.8965, Y 89.5499, Z -7.1667, A 0.000, B 0.000, C 0.000 }
gfCNCPoint5[12862] = {X 120.0690, Y 88.7328, Z -7.1667, A 0.000, B 0.000, C 0.000 }
gfCNCPoint5[12863] = {X 121.3491, Y 88.0972, Z -7.1667, A 0.000, B 0.000, C 0.000 }
gfCNCPoint5[12864] = {X 122.7089, Y 87.6570, Z -7.1667, A 0.000, B 0.000, C 0.000 }
gfCNCPoint5[12865] = {X 124.1186, Y 87.4219, Z -7.1667, A 0.000, B 0.000, C 0.000 }
gfCNCPoint5[12866] = {X 124.5382, Y 87.3596, Z -7.1667, A 0.000, B 0.000, C 0.000 }
gfCNCPoint5[12867] = {X 124.9951, Y 86.8921, Z -7.1667, A 0.000, B 0.000, C 0.000 }
gfCNCPoint5[12868] = {X 125.4394, Y 86.4125, Z -7.1667, A 0.000, B 0.000, C 0.000 }
gfCNCPoint5[12869] = {X 149.6584, Y 59.8183, Z -7.1667, A 0.000, B 0.000, C 0.000 }
gfCNCPoint5[12870] = {X 149.6295, Y 59.4061, Z -7.1667, A 0.000, B 0.000, C 0.000 }
gfCNCPoint5[12871] = {X 149.6181, Y 58.9930, Z -7.1667, A 0.000, B 0.000, C 0.000 }
gfCNCPoint5[12872] = {X 149.6180, Y 58.0000, Z -7.1667, A 0.000, B 0.000, C 0.000 }
gfCNCPoint5[12873] = {X 149.6915, Y 56.8093, Z -7.1667, A 0.000, B 0.000, C 0.000 }
gfCNCPoint5[12874] = {X 149.9109, Y 55.6367, Z -7.1667, A 0.000, B 0.000, C 0.000 }
gfCNCPoint5[12875] = {X 150.2729, Y 54.5000, Z -7.1667, A 0.000, B 0.000, C 0.000 }
gfCNCPoint5[12876] = {X 150.7719, Y 53.4164, Z -7.1667, A 0.000, B 0.000, C 0.000 }
gfCNCPoint5[12877] = {X 151.5117, Y 52.2488, Z -7.1667, A 0.000, B 0.000, C 0.000 }
gfCNCPoint5[12878] = {X 152.4103, Y 51.1984, Z -7.1667, A 0.000, B 0.000, C 0.000 }
gfCNCPoint5[12879] = {X 153.4493, Y 50.2867, Z -7.1667, A 0.000, B 0.000, C 0.000 }
gfCNCPoint5[12880] = {X 154.6075, Y 49.5323, Z -7.1667, A 0.000, B 0.000, C 0.000 }
gfCNCPoint5[12881] = {X 155.8614, Y 48.9505, Z -7.1667, A 0.000, B 0.000, C 0.000 }
gfCNCPoint5[12882] = {X 157.1854, Y 48.5533, Z -7.1667, A 0.000, B 0.000, C 0.000 }
gfCNCPoint5[12883] = {X 158.2353, Y 48.3785, Z -7.1667, A 0.000, B 0.000, C 0.000 }
gfCNCPoint5[12884] = {X 159.2980, Y 48.3200, Z -7.1667, A 0.000, B 0.000, C 0.000 }
gfCNCPoint5[12885] = {X 176.3014, Y 48.3200, Z -7.1667, A 0.000, B 0.000, C 0.000 }
gfCNCPoint5[12886] = {X 174.9297, Y 47.4865, Z -7.1667, A 0.000, B 0.000, C 0.000 }
gfCNCPoint5[12887] = {X 173.6419, Y 46.5284, Z -7.1667, A 0.000, B 0.000, C 0.000 }
gfCNCPoint5[12888] = {X 172.5421, Y 45.5341, Z -7.1667, A 0.000, B 0.000, C 0.000 }
gfCNCPoint5[12889] = {X 171.5572, Y 44.4259, Z -7.1667, A 0.000, B 0.000, C 0.000 }
gfCNCPoint5[12890] = {X 170.5958, Y 43.0508, Z -7.1667, A 0.000, B 0.000, C 0.000 }
gfCNCPoint5[12891] = {X 169.8111, Y 41.5676, Z -7.1667, A 0.000, B 0.000, C 0.000 }
gfCNCPoint5[12892] = {X 169.2152, Y 39.9990, Z -7.1667, A 0.000, B 0.000, C 0.000 }
gfCNCPoint5[12893] = {X 168.8173, Y 38.3690, Z -7.1667, A 0.000, B 0.000, C 0.000 }
gfCNCPoint5[12894] = {X 168.7070, Y 37.6766, Z -7.1667, A 0.000, B 0.000, C 0.000 }
gfCNCPoint5[12895] = {X 168.5425, Y 36.0107, Z -7.1667, A 0.000, B 0.000, C 0.000 }
gfCNCPoint5[12896] = {X 168.5599, Y 34.3367, Z -7.1667, A 0.000, B 0.000, C 0.000 }
gfCNCPoint5[12897] = {X 168.7591, Y 32.6746, Z -7.1667, A 0.000, B 0.000, C 0.000 }
gfCNCPoint5[12898] = {X 169.1378, Y 31.0439, Z -7.1667, A 0.000, B 0.000, C 0.000 }
gfCNCPoint5[12899] = {X 169.6914, Y 29.4640, Z -7.1667, A 0.000, B 0.000, C 0.000 }
gfCNCPoint5[12900] = {X 170.2632, Y 28.2672, Z -7.1667, A 0.000, B 0.000, C 0.000 }
gfCNCPoint5[12901] = {X 170.9700, Y 27.1448, Z -7.1667, A 0.000, B 0.000, C 0.000 }
gfCNCPoint5[12902] = {X 171.8022, Y 26.1120, Z -7.1667, A 0.000, B 0.000, C 0.000 }
gfCNCPoint5[12903] = {X 172.7486, Y 25.1827, Z -7.1667, A 0.000, B 0.000, C 0.000 }
gfCNCPoint5[12904] = {X 173.7965, Y 24.3695, Z -7.1667, A 0.000, B 0.000, C 0.000 }
gfCNCPoint5[12905] = {X 173.0266, Y 23.7513, Z -7.1667, A 0.000, B 0.000, C 0.000 }
gfCNCPoint5[12906] = {X 172.3970, Y 22.9909, Z -7.1667, A 0.000, B 0.000, C 0.000 }
gfCNCPoint5[12907] = {X 171.9332, Y 22.1193, Z -7.1667, A 0.000, B 0.000, C 0.000 }
gfCNCPoint5[12908] = {X 169.3220, Y 15.7237, Z -7.1667, A 0.000, B 0.000, C 0.000 }
gfCNCPoint5[12909] = {X 169.1088, Y 15.0753, Z -7.1667, A 0.000, B 0.000, C 0.000 }
gfCNCPoint5[12910] = {X 168.9882, Y 14.4035, Z -7.1667, A 0.000, B 0.000, C 0.000 }
gfCNCPoint5[12911] = {X 168.9599, Y 13.8791, Z -7.1667, A 0.000, B 0.000, C 0.000 }
gfCNCPoint5[12912] = {X 168.9882, Y 13.3548, Z -7.1667, A 0.000, B 0.000, C 0.000 }
gfCNCPoint5[12913] = {X 169.1590, Y 12.4995, Z -7.1667, A 0.000, B 0.000, C 0.000 }
gfCNCPoint5[12914] = {X 169.4794, Y 11.6882, Z -7.1667, A 0.000, B 0.000, C 0.000 }
gfCNCPoint5[12915] = {X 169.9391, Y 10.9469, Z -7.1667, A 0.000, B 0.000, C 0.000 }
gfCNCPoint5[12916] = {X 170.6136, Y 10.2178, Z -7.1667, A 0.000, B 0.000, C 0.000 }
gfCNCPoint5[12917] = {X 171.4217, Y 9.6404, Z -7.1667, A 0.000, B 0.000, C 0.000 }
gfCNCPoint5[12918] = {X 172.0576, Y 9.2779, Z -7.1667, A 0.000, B 0.000, C 0.000 }
gfCNCPoint5[12919] = {X 172.9924, Y 8.8772, Z -7.1667, A 0.000, B 0.000, C 0.000 }
gfCNCPoint5[12920] = {X 173.9900, Y 8.6790, Z -7.1667, A 0.000, B 0.000, C 0.000 }
gfCNCPoint5[12921] = {X 175.0071, Y 8.6919, Z -7.1667, A 0.000, B 0.000, C 0.000 }
gfCNCPoint5[12922] = {X 175.9993, Y 8.9153, Z -7.1667, A 0.000, B 0.000, C 0.000 }
gfCNCPoint5[12923] = {X 176.9087, Y 8.5286, Z -7.1667, A 0.000, B 0.000, C 0.000 }
gfCNCPoint5[12924] = {X 179.1572, Y 7.7024, Z -7.1667, A 0.000, B 0.000, C 0.000 }
gfCNCPoint5[12925] = {X 181.4771, Y 7.1049, Z -7.1667, A 0.000, B 0.000, C 0.000 }
gfCNCPoint5[12926] = {X 168.0206, Y 7.1049, Z -7.1667, A 0.000, B 0.000, C 0.000 }
gfCNCPoint5[12927] = {X 168.0206, Y 4.7049, Z -7.1667, A 0.000, B 0.000, C 0.000 }
gfCNCPoint5[12928] = {X 155.1592, Y 4.7049, Z -7.1667, A 0.000, B 0.000, C 0.000 }
gfCNCPoint5[12929] = {X 155.1592, Y 7.1049, Z -7.1667, A 0.000, B 0.000, C 0.000 }
gfCNCPoint5[12930] = {X 137.3635, Y 7.1049, Z -7.1667, A 0.000, B 0.000, C 0.000 }
gfCNCPoint5[12931] = {X 137.5330, Y 7.2909, Z -7.1667, A 0.000, B 0.000, C 0.000 }
gfCNCPoint5[12932] = {X 137.6927, Y 7.4854, Z -7.1667, A 0.000, B 0.000, C 0.000 }
gfCNCPoint5[12933] = {X 154.8300, Y 7.4854, Z -7.1667, A 0.000, B 0.000, C 0.000 }
gfCNCPoint5[12934] = {X 154.9897, Y 7.2909, Z -7.1667, A 0.000, B 0.000, C 0.000 }
gfCNCPoint5[12935] = {X 155.1592, Y 7.1049, Z -7.1667, A 0.000, B 0.000, C 0.000 }
gfCNCPoint5[12936] = {X 155.1592, Y 4.7049, Z -7.1667, A 0.000, B 0.000, C 0.000 }
gfCNCPoint5[12937] = {X 42.6032, Y 4.7049, Z -7.1667, A 0.000, B 0.000, C 0.000 }
gfCNCPoint5[12938] = {X 42.6032, Y 9.5049, Z -7.1667, A 0.000, B 0.000, C 0.000 }
gfCNCPoint5[12939] = {X 36.0465, Y 9.5049, Z -7.1667, A 0.000, B 0.000, C 0.000 }
gfCNCPoint5[12940] = {X 37.0565, Y 11.3879, Z -7.1667, A 0.000, B 0.000, C 0.000 }
gfCNCPoint5[12941] = {X 37.8848, Y 13.3577, Z -7.1667, A 0.000, B 0.000, C 0.000 }
gfCNCPoint5[12942] = {X 38.5472, Y 15.5381, Z -7.1667, A 0.000, B 0.000, C 0.000 }
gfCNCPoint5[12943] = {X 39.0058, Y 17.7703, Z -7.1667, A 0.000, B 0.000, C 0.000 }
gfCNCPoint5[12944] = {X 39.2565, Y 20.0353, Z -7.1667, A 0.000, B 0.000, C 0.000 }
gfCNCPoint5[12945] = {X 39.2973, Y 22.3138, Z -7.1667, A 0.000, B 0.000, C 0.000 }
gfCNCPoint5[12946] = {X 39.1277, Y 24.5863, Z -7.1667, A 0.000, B 0.000, C 0.000 }
gfCNCPoint5[12947] = {X 42.5393, Y 15.4278, Z -7.1667, A 0.000, B 0.000, C 0.000 }
gfCNCPoint5[12948] = {X 42.3081, Y 14.2496, Z -7.1667, A 0.000, B 0.000, C 0.000 }
gfCNCPoint5[12949] = {X 42.2245, Y 13.0518, Z -7.1667, A 0.000, B 0.000, C 0.000 }
gfCNCPoint5[12950] = {X 42.2242, Y 12.1868, Z -7.1667, A 0.000, B 0.000, C 0.000 }
gfCNCPoint5[12951] = {X 42.3194, Y 10.8325, Z -7.1667, A 0.000, B 0.000, C 0.000 }
gfCNCPoint5[12952] = {X 42.6032, Y 9.5049, Z -7.1667, A 0.000, B 0.000, C 0.000 }
gfCNCPoint5[12953] = {X 42.6032, Y 7.1049, Z -7.1667, A 0.000, B 0.000, C 0.000 }
gfCNCPoint5[12954] = {X 31.2121, Y 7.1049, Z -7.1667, A 0.000, B 0.000, C 0.000 }
gfCNCPoint5[12955] = {X 32.2275, Y 8.2449, Z -7.1667, A 0.000, B 0.000, C 0.000 }
gfCNCPoint5[12956] = {X 33.1543, Y 9.4581, Z -7.1667, A 0.000, B 0.000, C 0.000 }
gfCNCPoint5[12957] = {X 33.9873, Y 10.7376, Z -7.1667, A 0.000, B 0.000, C 0.000 }
gfCNCPoint5[12958] = {X 34.8879, Y 12.4162, Z -7.1667, A 0.000, B 0.000, C 0.000 }
gfCNCPoint5[12959] = {X 35.6271, Y 14.1718, Z -7.1667, A 0.000, B 0.000, C 0.000 }
gfCNCPoint5[12960] = {X 36.2235, Y 16.1382, Z -7.1667, A 0.000, B 0.000, C 0.000 }
gfCNCPoint5[12961] = {X 36.6362, Y 18.1512, Z -7.1667, A 0.000, B 0.000, C 0.000 }
gfCNCPoint5[12962] = {X 36.8617, Y 20.1937, Z -7.1667, A 0.000, B 0.000, C 0.000 }
gfCNCPoint5[12963] = {X 36.8981, Y 22.2482, Z -7.1667, A 0.000, B 0.000, C 0.000 }
gfCNCPoint5[12964] = {X 36.7452, Y 24.2974, Z -7.1667, A 0.000, B 0.000, C 0.000 }
gfCNCPoint5[12965] = {X 36.5519, Y 25.5789, Z -7.1667, A 0.000, B 0.000, C 0.000 }
gfCNCPoint5[12966] = {X 36.2844, Y 26.8469, Z -7.1667, A 0.000, B 0.000, C 0.000 }
gfCNCPoint5[12967] = {X 35.8753, Y 28.3065, Z -7.1667, A 0.000, B 0.000, C 0.000 }
gfCNCPoint5[12968] = {X 35.3510, Y 29.7288, Z -7.1667, A 0.000, B 0.000, C 0.000 }
gfCNCPoint5[12969] = {X 34.7149, Y 31.1047, Z -7.1667, A 0.000, B 0.000, C 0.000 }
gfCNCPoint5[12970] = {X 37.2838, Y 36.4117, Z -7.1667, A 0.000, B 0.000, C 0.000 }
gfCNCPoint5[12971] = {X 41.3767, Y 25.4240, Z -7.1667, A 0.000, B 0.000, C 0.000 }
gfCNCPoint5[12972] = {X 45.0743, Y 15.4980, Z -7.1667, A 0.000, B 0.000, C 0.000 }
gfCNCPoint5[12973] = {X 44.7425, Y 14.2852, Z -7.1667, A 0.000, B 0.000, C 0.000 }
gfCNCPoint5[12974] = {X 44.6244, Y 13.0334, Z -7.1667, A 0.000, B 0.000, C 0.000 }
gfCNCPoint5[12975] = {X 44.6242, Y 12.1868, Z -7.1667, A 0.000, B 0.000, C 0.000 }
gfCNCPoint5[12976] = {X 44.6958, Y 11.1683, Z -7.1667, A 0.000, B 0.000, C 0.000 }
gfCNCPoint5[12977] = {X 44.9092, Y 10.1698, Z -7.1667, A 0.000, B 0.000, C 0.000 }
gfCNCPoint5[12978] = {X 45.3323, Y 9.0549, Z -7.1667, A 0.000, B 0.000, C 0.000 }
gfCNCPoint5[12979] = {X 45.9318, Y 8.0240, Z -7.1667, A 0.000, B 0.000, C 0.000 }
gfCNCPoint5[12980] = {X 46.6915, Y 7.1049, Z -7.1667, A 0.000, B 0.000, C 0.000 }
gfCNCPoint5[12981] = {X 42.6032, Y 7.1049, Z -7.1667, A 0.000, B 0.000, C 0.000 }
gfCNCPoint5[12982] = {X 42.6032, Y 4.7049, Z -7.1667, A 0.000, B 0.000, C 0.000 }
gfCNCPoint5[12983] = {X 23.8370, Y 4.7049, Z -7.1667, A 0.000, B 0.000, C 0.000 }
gfCNCPoint5[12984] = {X 25.7645, Y 5.7846, Z -7.1667, A 0.000, B 0.000, C 0.000 }
gfCNCPoint5[12985] = {X 27.5759, Y 7.0495, Z -7.1667, A 0.000, B 0.000, C 0.000 }
gfCNCPoint5[12986] = {X 28.5594, Y 7.8743, Z -7.1667, A 0.000, B 0.000, C 0.000 }
gfCNCPoint5[12987] = {X 29.4813, Y 8.7674, Z -7.1667, A 0.000, B 0.000, C 0.000 }
gfCNCPoint5[12988] = {X 30.6895, Y 10.1628, Z -7.1667, A 0.000, B 0.000, C 0.000 }
gfCNCPoint5[12989] = {X 31.7475, Y 11.6752, Z -7.1667, A 0.000, B 0.000, C 0.000 }
gfCNCPoint5[12990] = {X 32.6439, Y 13.2887, Z -7.1667, A 0.000, B 0.000, C 0.000 }
gfCNCPoint5[12991] = {X 33.3693, Y 14.9859, Z -7.1667, A 0.000, B 0.000, C 0.000 }
gfCNCPoint5[12992] = {X 33.9194, Y 16.8169, Z -7.1667, A 0.000, B 0.000, C 0.000 }
gfCNCPoint5[12993] = {X 34.2910, Y 18.6923, Z -7.1667, A 0.000, B 0.000, C 0.000 }
gfCNCPoint5[12994] = {X 34.4809, Y 20.5946, Z -7.1667, A 0.000, B 0.000, C 0.000 }
gfCNCPoint5[12995] = {X 34.4872, Y 22.5064, Z -7.1667, A 0.000, B 0.000, C 0.000 }
gfCNCPoint5[12996] = {X 34.3098, Y 24.4100, Z -7.1667, A 0.000, B 0.000, C 0.000 }
gfCNCPoint5[12997] = {X 33.9504, Y 26.2878, Z -7.1667, A 0.000, B 0.000, C 0.000 }
gfCNCPoint5[12998] = {X 33.4665, Y 27.9396, Z -7.1667, A 0.000, B 0.000, C 0.000 }
gfCNCPoint5[12999] = {X 32.8139, Y 29.5324, Z -7.1667, A 0.000, B 0.000, C 0.000 }
gfCNCPoint5[13000] = {X 31.9995, Y 31.0489, Z -7.1667, A 0.000, B 0.000, C 0.000 }
gfCNCPoint5[13001] = {X 32.1288, Y 31.2843, Z -7.1667, A 0.000, B 0.000, C 0.000 }
gfCNCPoint5[13002] = {X 32.2511, Y 31.5234, Z -7.1667, A 0.000, B 0.000, C 0.000 }
gfCNCPoint5[13003] = {X 35.3025, Y 37.8269, Z -7.1667, A 0.000, B 0.000, C 0.000 }
gfCNCPoint5[13004] = {X 35.7263, Y 38.8573, Z -7.1667, A 0.000, B 0.000, C 0.000 }
gfCNCPoint5[13005] = {X 36.0224, Y 39.9313, Z -7.1667, A 0.000, B 0.000, C 0.000 }
gfCNCPoint5[13006] = {X 36.1865, Y 41.0332, Z -7.1667, A 0.000, B 0.000, C 0.000 }
gfCNCPoint5[13007] = {X 36.2163, Y 42.1469, Z -7.1667, A 0.000, B 0.000, C 0.000 }
gfCNCPoint5[13008] = {X 36.6302, Y 41.4265, Z -7.1667, A 0.000, B 0.000, C 0.000 }
gfCNCPoint5[13009] = {X 37.1603, Y 40.7867, Z -7.1667, A 0.000, B 0.000, C 0.000 }
gfCNCPoint5[13010] = {X 37.7913, Y 40.2461, Z -7.1667, A 0.000, B 0.000, C 0.000 }
gfCNCPoint5[13011] = {X 38.5048, Y 39.8204, Z -7.1667, A 0.000, B 0.000, C 0.000 }
gfCNCPoint5[13012] = {X 39.0436, Y 38.5343, Z -7.1667, A 0.000, B 0.000, C 0.000 }
gfCNCPoint5[13013] = {X 39.5396, Y 37.2311, Z -7.1667, A 0.000, B 0.000, C 0.000 }
gfCNCPoint5[13014] = {X 47.6702, Y 15.4045, Z -7.1667, A 0.000, B 0.000, C 0.000 }
gfCNCPoint5[13015] = {X 47.3200, Y 14.6512, Z -7.1667, A 0.000, B 0.000, C 0.000 }
gfCNCPoint5[13016] = {X 47.1026, Y 13.8493, Z -7.1667, A 0.000, B 0.000, C 0.000 }
gfCNCPoint5[13017] = {X 47.0244, Y 13.0222, Z -7.1667, A 0.000, B 0.000, C 0.000 }
gfCNCPoint5[13018] = {X 47.0242, Y 12.1868, Z -7.1667, A 0.000, B 0.000, C 0.000 }
gfCNCPoint5[13019] = {X 47.1150, Y 11.2500, Z -7.1667, A 0.000, B 0.000, C 0.000 }
gfCNCPoint5[13020] = {X 47.3839, Y 10.3480, Z -7.1667, A 0.000, B 0.000, C 0.000 }
gfCNCPoint5[13021] = {X 47.8210, Y 9.5144, Z -7.1667, A 0.000, B 0.000, C 0.000 }
gfCNCPoint5[13022] = {X 48.4100, Y 8.7802, Z -7.1667, A 0.000, B 0.000, C 0.000 }
gfCNCPoint5[13023] = {X 49.1545, Y 8.1552, Z -7.1667, A 0.000, B 0.000, C 0.000 }
gfCNCPoint5[13024] = {X 50.0081, Y 7.6902, Z -7.1667, A 0.000, B 0.000, C 0.000 }
gfCNCPoint5[13025] = {X 50.9370, Y 7.4036, Z -7.1667, A 0.000, B 0.000, C 0.000 }
gfCNCPoint5[13026] = {X 51.9042, Y 7.3068, Z -7.1667, A 0.000, B 0.000, C 0.000 }
gfCNCPoint5[13027] = {X 59.6221, Y 7.3068, Z -7.1667, A 0.000, B 0.000, C 0.000 }
gfCNCPoint5[13028] = {X 60.5894, Y 7.4036, Z -7.1667, A 0.000, B 0.000, C 0.000 }
gfCNCPoint5[13029] = {X 61.5182, Y 7.6902, Z -7.1667, A 0.000, B 0.000, C 0.000 }
gfCNCPoint5[13030] = {X 62.3718, Y 8.1552, Z -7.1667, A 0.000, B 0.000, C 0.000 }
gfCNCPoint5[13031] = {X 63.1163, Y 8.7802, Z -7.1667, A 0.000, B 0.000, C 0.000 }
gfCNCPoint5[13032] = {X 63.7053, Y 9.5144, Z -7.1667, A 0.000, B 0.000, C 0.000 }
gfCNCPoint5[13033] = {X 64.1424, Y 10.3480, Z -7.1667, A 0.000, B 0.000, C 0.000 }
gfCNCPoint5[13034] = {X 64.4114, Y 11.2500, Z -7.1667, A 0.000, B 0.000, C 0.000 }
gfCNCPoint5[13035] = {X 64.5021, Y 12.1868, Z -7.1667, A 0.000, B 0.000, C 0.000 }
gfCNCPoint5[13036] = {X 64.5019, Y 13.0237, Z -7.1667, A 0.000, B 0.000, C 0.000 }
gfCNCPoint5[13037] = {X 64.4205, Y 13.8670, Z -7.1667, A 0.000, B 0.000, C 0.000 }
gfCNCPoint5[13038] = {X 64.1944, Y 14.6835, Z -7.1667, A 0.000, B 0.000, C 0.000 }
gfCNCPoint5[13039] = {X 63.8305, Y 15.4486, Z -7.1667, A 0.000, B 0.000, C 0.000 }
gfCNCPoint5[13040] = {X 72.9557, Y 39.8585, Z -7.1667, A 0.000, B 0.000, C 0.000 }
gfCNCPoint5[13041] = {X 73.8453, Y 40.4406, Z -7.1667, A 0.000, B 0.000, C 0.000 }
gfCNCPoint5[13042] = {X 74.5877, Y 41.2014, Z -7.1667, A 0.000, B 0.000, C 0.000 }
gfCNCPoint5[13043] = {X 75.1477, Y 42.1050, Z -7.1667, A 0.000, B 0.000, C 0.000 }
gfCNCPoint5[13044] = {X 75.4988, Y 43.1084, Z -7.1667, A 0.000, B 0.000, C 0.000 }
gfCNCPoint5[13045] = {X 75.6243, Y 44.1640, Z -7.1667, A 0.000, B 0.000, C 0.000 }
gfCNCPoint5[13046] = {X 75.6245, Y 45.0000, Z -7.1667, A 0.000, B 0.000, C 0.000 }
gfCNCPoint5[13047] = {X 75.5307, Y 45.9520, Z -7.1667, A 0.000, B 0.000, C 0.000 }
gfCNCPoint5[13048] = {X 75.2530, Y 46.8675, Z -7.1667, A 0.000, B 0.000, C 0.000 }
gfCNCPoint5[13049] = {X 74.8020, Y 47.7112, Z -7.1667, A 0.000, B 0.000, C 0.000 }
gfCNCPoint5[13050] = {X 74.1951, Y 48.4507, Z -7.1667, A 0.000, B 0.000, C 0.000 }
gfCNCPoint5[13051] = {X 73.4556, Y 49.0576, Z -7.1667, A 0.000, B 0.000, C 0.000 }
gfCNCPoint5[13052] = {X 72.6120, Y 49.5085, Z -7.1667, A 0.000, B 0.000, C 0.000 }
gfCNCPoint5[13053] = {X 71.6965, Y 49.7862, Z -7.1667, A 0.000, B 0.000, C 0.000 }
gfCNCPoint5[13054] = {X 70.7445, Y 49.8800, Z -7.1667, A 0.000, B 0.000, C 0.000 }
gfCNCPoint5[13055] = {X 64.1851, Y 49.8800, Z -7.1667, A 0.000, B 0.000, C 0.000 }
gfCNCPoint5[13056] = {X 63.2331, Y 49.7862, Z -7.1667, A 0.000, B 0.000, C 0.000 }
gfCNCPoint5[13057] = {X 62.3176, Y 49.5085, Z -7.1667, A 0.000, B 0.000, C 0.000 }
gfCNCPoint5[13058] = {X 61.4740, Y 49.0576, Z -7.1667, A 0.000, B 0.000, C 0.000 }
gfCNCPoint5[13059] = {X 60.7345, Y 48.4507, Z -7.1667, A 0.000, B 0.000, C 0.000 }
gfCNCPoint5[13060] = {X 60.1276, Y 47.7112, Z -7.1667, A 0.000, B 0.000, C 0.000 }
gfCNCPoint5[13061] = {X 59.6766, Y 46.8675, Z -7.1667, A 0.000, B 0.000, C 0.000 }
gfCNCPoint5[13062] = {X 59.3989, Y 45.9520, Z -7.1667, A 0.000, B 0.000, C 0.000 }
gfCNCPoint5[13063] = {X 59.3051, Y 45.0000, Z -7.1667, A 0.000, B 0.000, C 0.000 }
gfCNCPoint5[13064] = {X 59.3052, Y 44.2028, Z -7.1667, A 0.000, B 0.000, C 0.000 }
gfCNCPoint5[13065] = {X 59.3847, Y 43.3314, Z -7.1667, A 0.000, B 0.000, C 0.000 }
gfCNCPoint5[13066] = {X 59.6185, Y 42.4882, Z -7.1667, A 0.000, B 0.000, C 0.000 }
gfCNCPoint5[13067] = {X 59.9992, Y 41.7003, Z -7.1667, A 0.000, B 0.000, C 0.000 }
gfCNCPoint5[13068] = {X 59.6150, Y 40.6492, Z -7.1667, A 0.000, B 0.000, C 0.000 }
gfCNCPoint5[13069] = {X 52.4673, Y 40.6492, Z -7.1667, A 0.000, B 0.000, C 0.000 }
gfCNCPoint5[13070] = {X 51.9475, Y 42.0460, Z -7.1667, A 0.000, B 0.000, C 0.000 }
gfCNCPoint5[13071] = {X 52.2219, Y 42.7250, Z -7.1667, A 0.000, B 0.000, C 0.000 }
gfCNCPoint5[13072] = {X 52.3916, Y 43.4374, Z -7.1667, A 0.000, B 0.000, C 0.000 }
gfCNCPoint5[13073] = {X 52.4528, Y 44.1672, Z -7.1667, A 0.000, B 0.000, C 0.000 }
gfCNCPoint5[13074] = {X 52.4529, Y 45.0000, Z -7.1667, A 0.000, B 0.000, C 0.000 }
gfCNCPoint5[13075] = {X 52.3592, Y 45.9520, Z -7.1667, A 0.000, B 0.000, C 0.000 }
gfCNCPoint5[13076] = {X 52.0815, Y 46.8675, Z -7.1667, A 0.000, B 0.000, C 0.000 }
gfCNCPoint5[13077] = {X 51.6305, Y 47.7112, Z -7.1667, A 0.000, B 0.000, C 0.000 }
gfCNCPoint5[13078] = {X 51.0236, Y 48.4507, Z -7.1667, A 0.000, B 0.000, C 0.000 }
gfCNCPoint5[13079] = {X 50.2841, Y 49.0576, Z -7.1667, A 0.000, B 0.000, C 0.000 }
gfCNCPoint5[13080] = {X 49.4404, Y 49.5085, Z -7.1667, A 0.000, B 0.000, C 0.000 }
gfCNCPoint5[13081] = {X 48.5250, Y 49.7862, Z -7.1667, A 0.000, B 0.000, C 0.000 }
gfCNCPoint5[13082] = {X 47.5729, Y 49.8800, Z -7.1667, A 0.000, B 0.000, C 0.000 }
gfCNCPoint5[13083] = {X 40.6393, Y 49.8800, Z -7.1667, A 0.000, B 0.000, C 0.000 }
gfCNCPoint5[13084] = {X 39.6433, Y 49.7773, Z -7.1667, A 0.000, B 0.000, C 0.000 }
gfCNCPoint5[13085] = {X 38.6892, Y 49.4734, Z -7.1667, A 0.000, B 0.000, C 0.000 }
gfCNCPoint5[13086] = {X 37.8173, Y 48.9813, Z -7.1667, A 0.000, B 0.000, C 0.000 }
gfCNCPoint5[13087] = {X 37.0641, Y 48.3215, Z -7.1667, A 0.000, B 0.000, C 0.000 }
gfCNCPoint5[13088] = {X 36.5085, Y 47.5983, Z -7.1667, A 0.000, B 0.000, C 0.000 }
gfCNCPoint5[13089] = {X 36.0972, Y 46.7843, Z -7.1667, A 0.000, B 0.000, C 0.000 }
gfCNCPoint5[13090] = {X 35.8445, Y 45.9080, Z -7.1667, A 0.000, B 0.000, C 0.000 }
gfCNCPoint5[13091] = {X 35.7593, Y 45.0000, Z -7.1667, A 0.000, B 0.000, C 0.000 }
gfCNCPoint5[13092] = {X 35.7593, Y 44.7148, Z -7.1667, A 0.000, B 0.000, C 0.000 }
gfCNCPoint5[13093] = {X 36.2393, Y 44.7148, Z -7.1667, A 0.000, B 0.000, C 0.000 }
gfCNCPoint5[13094] = {X 36.2397, Y 44.1483, Z -7.1667, A 0.000, B 0.000, C 0.000 }
gfCNCPoint5[13095] = {X 36.3680, Y 43.1524, Z -7.1667, A 0.000, B 0.000, C 0.000 }
gfCNCPoint5[13096] = {X 36.7187, Y 42.2116, Z -7.1667, A 0.000, B 0.000, C 0.000 }
gfCNCPoint5[13097] = {X 37.2735, Y 41.3748, Z -7.1667, A 0.000, B 0.000, C 0.000 }
gfCNCPoint5[13098] = {X 38.0036, Y 40.6856, Z -7.1667, A 0.000, B 0.000, C 0.000 }
gfCNCPoint5[13099] = {X 38.8709, Y 40.1798, Z -7.1667, A 0.000, B 0.000, C 0.000 }
gfCNCPoint5[13100] = {X 39.4545, Y 38.7990, Z -7.1667, A 0.000, B 0.000, C 0.000 }
gfCNCPoint5[13101] = {X 39.9894, Y 37.3986, Z -7.1667, A 0.000, B 0.000, C 0.000 }
gfCNCPoint5[13102] = {X 48.2011, Y 15.3544, Z -7.1667, A 0.000, B 0.000, C 0.000 }
gfCNCPoint5[13103] = {X 47.8187, Y 14.6115, Z -7.1667, A 0.000, B 0.000, C 0.000 }
gfCNCPoint5[13104] = {X 47.5835, Y 13.8097, Z -7.1667, A 0.000, B 0.000, C 0.000 }
gfCNCPoint5[13105] = {X 47.5042, Y 12.9780, Z -7.1667, A 0.000, B 0.000, C 0.000 }
gfCNCPoint5[13106] = {X 47.5042, Y 12.1868, Z -7.1667, A 0.000, B 0.000, C 0.000 }
gfCNCPoint5[13107] = {X 47.6145, Y 11.2077, Z -7.1667, A 0.000, B 0.000, C 0.000 }
gfCNCPoint5[13108] = {X 47.9400, Y 10.2777, Z -7.1667, A 0.000, B 0.000, C 0.000 }
gfCNCPoint5[13109] = {X 48.4642, Y 9.4435, Z -7.1667, A 0.000, B 0.000, C 0.000 }
gfCNCPoint5[13110] = {X 49.1609, Y 8.7468, Z -7.1667, A 0.000, B 0.000, C 0.000 }
gfCNCPoint5[13111] = {X 49.9951, Y 8.2226, Z -7.1667, A 0.000, B 0.000, C 0.000 }
gfCNCPoint5[13112] = {X 50.9251, Y 7.8971, Z -7.1667, A 0.000, B 0.000, C 0.000 }
gfCNCPoint5[13113] = {X 51.9042, Y 7.7868, Z -7.1667, A 0.000, B 0.000, C 0.000 }
gfCNCPoint5[13114] = {X 59.6221, Y 7.7868, Z -7.1667, A 0.000, B 0.000, C 0.000 }
gfCNCPoint5[13115] = {X 60.6012, Y 7.8971, Z -7.1667, A 0.000, B 0.000, C 0.000 }
gfCNCPoint5[13116] = {X 61.5312, Y 8.2226, Z -7.1667, A 0.000, B 0.000, C 0.000 }
gfCNCPoint5[13117] = {X 62.3655, Y 8.7468, Z -7.1667, A 0.000, B 0.000, C 0.000 }
gfCNCPoint5[13118] = {X 63.0622, Y 9.4435, Z -7.1667, A 0.000, B 0.000, C 0.000 }
gfCNCPoint5[13119] = {X 63.5864, Y 10.2777, Z -7.1667, A 0.000, B 0.000, C 0.000 }
gfCNCPoint5[13120] = {X 63.9118, Y 11.2077, Z -7.1667, A 0.000, B 0.000, C 0.000 }
gfCNCPoint5[13121] = {X 64.0221, Y 12.1868, Z -7.1667, A 0.000, B 0.000, C 0.000 }
gfCNCPoint5[13122] = {X 64.0219, Y 13.0233, Z -7.1667, A 0.000, B 0.000, C 0.000 }
gfCNCPoint5[13123] = {X 63.9336, Y 13.8560, Z -7.1667, A 0.000, B 0.000, C 0.000 }
gfCNCPoint5[13124] = {X 63.6892, Y 14.6569, Z -7.1667, A 0.000, B 0.000, C 0.000 }
gfCNCPoint5[13125] = {X 63.2975, Y 15.3970, Z -7.1667, A 0.000, B 0.000, C 0.000 }
gfCNCPoint5[13126] = {X 63.5018, Y 15.9354, Z -7.1667, A 0.000, B 0.000, C 0.000 }
gfCNCPoint5[13127] = {X 66.3154, Y 23.4029, Z -7.1667, A 0.000, B 0.000, C 0.000 }
gfCNCPoint5[13128] = {X 72.2854, Y 39.4717, Z -7.1667, A 0.000, B 0.000, C 0.000 }
gfCNCPoint5[13129] = {X 72.5786, Y 40.2093, Z -7.1667, A 0.000, B 0.000, C 0.000 }
gfCNCPoint5[13130] = {X 73.4357, Y 40.7278, Z -7.1667, A 0.000, B 0.000, C 0.000 }
gfCNCPoint5[13131] = {X 74.1533, Y 41.4268, Z -7.1667, A 0.000, B 0.000, C 0.000 }
gfCNCPoint5[13132] = {X 74.6943, Y 42.2700, Z -7.1667, A 0.000, B 0.000, C 0.000 }
gfCNCPoint5[13133] = {X 75.0304, Y 43.2136, Z -7.1667, A 0.000, B 0.000, C 0.000 }
gfCNCPoint5[13134] = {X 75.1445, Y 44.2089, Z -7.1667, A 0.000, B 0.000, C 0.000 }
gfCNCPoint5[13135] = {X 75.1445, Y 45.0000, Z -7.1667, A 0.000, B 0.000, C 0.000 }
gfCNCPoint5[13136] = {X 75.0341, Y 45.9791, Z -7.1667, A 0.000, B 0.000, C 0.000 }
gfCNCPoint5[13137] = {X 74.7087, Y 46.9091, Z -7.1667, A 0.000, B 0.000, C 0.000 }
gfCNCPoint5[13138] = {X 74.1845, Y 47.7434, Z -7.1667, A 0.000, B 0.000, C 0.000 }
gfCNCPoint5[13139] = {X 73.4878, Y 48.4401, Z -7.1667, A 0.000, B 0.000, C 0.000 }
gfCNCPoint5[13140] = {X 72.6535, Y 48.9643, Z -7.1667, A 0.000, B 0.000, C 0.000 }
gfCNCPoint5[13141] = {X 71.7236, Y 49.2897, Z -7.1667, A 0.000, B 0.000, C 0.000 }
gfCNCPoint5[13142] = {X 70.7445, Y 49.4000, Z -7.1667, A 0.000, B 0.000, C 0.000 }
gfCNCPoint5[13143] = {X 64.1851, Y 49.4000, Z -7.1667, A 0.000, B 0.000, C 0.000 }
gfCNCPoint5[13144] = {X 63.2060, Y 49.2897, Z -7.1667, A 0.000, B 0.000, C 0.000 }
gfCNCPoint5[13145] = {X 62.2760, Y 48.9643, Z -7.1667, A 0.000, B 0.000, C 0.000 }
gfCNCPoint5[13146] = {X 61.4418, Y 48.4401, Z -7.1667, A 0.000, B 0.000, C 0.000 }
gfCNCPoint5[13147] = {X 60.7451, Y 47.7434, Z -7.1667, A 0.000, B 0.000, C 0.000 }
gfCNCPoint5[13148] = {X 60.2209, Y 46.9091, Z -7.1667, A 0.000, B 0.000, C 0.000 }
gfCNCPoint5[13149] = {X 59.8955, Y 45.9791, Z -7.1667, A 0.000, B 0.000, C 0.000 }
gfCNCPoint5[13150] = {X 59.7851, Y 45.0000, Z -7.1667, A 0.000, B 0.000, C 0.000 }
gfCNCPoint5[13151] = {X 59.7856, Y 44.1483, Z -7.1667, A 0.000, B 0.000, C 0.000 }
gfCNCPoint5[13152] = {X 59.8783, Y 43.3082, Z -7.1667, A 0.000, B 0.000, C 0.000 }
gfCNCPoint5[13153] = {X 60.1299, Y 42.5014, Z -7.1667, A 0.000, B 0.000, C 0.000 }
gfCNCPoint5[13154] = {X 60.5312, Y 41.7575, Z -7.1667, A 0.000, B 0.000, C 0.000 }
gfCNCPoint5[13155] = {X 59.9506, Y 40.1692, Z -7.1667, A 0.000, B 0.000, C 0.000 }
gfCNCPoint5[13156] = {X 52.1338, Y 40.1692, Z -7.1667, A 0.000, B 0.000, C 0.000 }
gfCNCPoint5[13157] = {X 51.4231, Y 42.0789, Z -7.1667, A 0.000, B 0.000, C 0.000 }
gfCNCPoint5[13158] = {X 51.7256, Y 42.7545, Z -7.1667, A 0.000, B 0.000, C 0.000 }
gfCNCPoint5[13159] = {X 51.9107, Y 43.4712, Z -7.1667, A 0.000, B 0.000, C 0.000 }
gfCNCPoint5[13160] = {X 51.9729, Y 44.2089, Z -7.1667, A 0.000, B 0.000, C 0.000 }
gfCNCPoint5[13161] = {X 51.9729, Y 45.0000, Z -7.1667, A 0.000, B 0.000, C 0.000 }
gfCNCPoint5[13162] = {X 51.8626, Y 45.9791, Z -7.1667, A 0.000, B 0.000, C 0.000 }
gfCNCPoint5[13163] = {X 51.5372, Y 46.9091, Z -7.1667, A 0.000, B 0.000, C 0.000 }
gfCNCPoint5[13164] = {X 51.0130, Y 47.7434, Z -7.1667, A 0.000, B 0.000, C 0.000 }
gfCNCPoint5[13165] = {X 50.3163, Y 48.4401, Z -7.1667, A 0.000, B 0.000, C 0.000 }
gfCNCPoint5[13166] = {X 49.4820, Y 48.9643, Z -7.1667, A 0.000, B 0.000, C 0.000 }
gfCNCPoint5[13167] = {X 48.5520, Y 49.2897, Z -7.1667, A 0.000, B 0.000, C 0.000 }
gfCNCPoint5[13168] = {X 47.5729, Y 49.4000, Z -7.1667, A 0.000, B 0.000, C 0.000 }
gfCNCPoint5[13169] = {X 40.6393, Y 49.4000, Z -7.1667, A 0.000, B 0.000, C 0.000 }
gfCNCPoint5[13170] = {X 39.6602, Y 49.2897, Z -7.1667, A 0.000, B 0.000, C 0.000 }
gfCNCPoint5[13171] = {X 38.7302, Y 48.9643, Z -7.1667, A 0.000, B 0.000, C 0.000 }
gfCNCPoint5[13172] = {X 37.8959, Y 48.4401, Z -7.1667, A 0.000, B 0.000, C 0.000 }
gfCNCPoint5[13173] = {X 37.1992, Y 47.7434, Z -7.1667, A 0.000, B 0.000, C 0.000 }
gfCNCPoint5[13174] = {X 36.6750, Y 46.9091, Z -7.1667, A 0.000, B 0.000, C 0.000 }
gfCNCPoint5[13175] = {X 36.3496, Y 45.9791, Z -7.1667, A 0.000, B 0.000, C 0.000 }
gfCNCPoint5[13176] = {X 36.2393, Y 45.0000, Z -7.1667, A 0.000, B 0.000, C 0.000 }
gfCNCPoint5[13177] = {X 36.2393, Y 44.7148, Z -7.1667, A 0.000, B 0.000, C 0.000 }
gfCNCPoint5[13178] = {X 35.7593, Y 44.7148, Z -7.1667, A 0.000, B 0.000, C 0.000 }
gfCNCPoint5[13179] = {X 35.2211, Y 46.0074, Z -7.1667, A 0.000, B 0.000, C 0.000 }
gfCNCPoint5[13180] = {X 34.4930, Y 47.2034, Z -7.1667, A 0.000, B 0.000, C 0.000 }
gfCNCPoint5[13181] = {X 33.5918, Y 48.2750, Z -7.1667, A 0.000, B 0.000, C 0.000 }
gfCNCPoint5[13182] = {X 33.2092, Y 48.6435, Z -7.1667, A 0.000, B 0.000, C 0.000 }
gfCNCPoint5[13183] = {X 32.8060, Y 48.9892, Z -7.1667, A 0.000, B 0.000, C 0.000 }
gfCNCPoint5[13184] = {X 32.2708, Y 49.4219, Z -7.1667, A 0.000, B 0.000, C 0.000 }
gfCNCPoint5[13185] = {X 31.1844, Y 50.1784, Z -7.1667, A 0.000, B 0.000, C 0.000 }
gfCNCPoint5[13186] = {X 30.0008, Y 50.7713, Z -7.1667, A 0.000, B 0.000, C 0.000 }
gfCNCPoint5[13187] = {X 28.7444, Y 51.1883, Z -7.1667, A 0.000, B 0.000, C 0.000 }
gfCNCPoint5[13188] = {X 27.4412, Y 51.4210, Z -7.1667, A 0.000, B 0.000, C 0.000 }
gfCNCPoint5[13189] = {X 26.1181, Y 51.4644, Z -7.1667, A 0.000, B 0.000, C 0.000 }
gfCNCPoint5[13190] = {X 23.6766, Y 52.5843, Z -7.1667, A 0.000, B 0.000, C 0.000 }
gfCNCPoint5[13191] = {X 21.1546, Y 53.5085, Z -7.1667, A 0.000, B 0.000, C 0.000 }
gfCNCPoint5[13192] = {X 18.9436, Y 54.1370, Z -7.1667, A 0.000, B 0.000, C 0.000 }
gfCNCPoint5[13193] = {X 16.6880, Y 54.5797, Z -7.1667, A 0.000, B 0.000, C 0.000 }
gfCNCPoint5[13194] = {X 14.4035, Y 54.8334, Z -7.1667, A 0.000, B 0.000, C 0.000 }
gfCNCPoint5[13195] = {X 12.1058, Y 54.8964, Z -7.1667, A 0.000, B 0.000, C 0.000 }
gfCNCPoint5[13196] = {X 9.8108, Y 54.7682, Z -7.1667, A 0.000, B 0.000, C 0.000 }
gfCNCPoint5[13197] = {X 7.5344, Y 54.4497, Z -7.1667, A 0.000, B 0.000, C 0.000 }
gfCNCPoint5[13198] = {X 7.1095, Y 54.3687, Z -7.1667, A 0.000, B 0.000, C 0.000 }
gfCNCPoint5[13199] = {X 6.6859, Y 54.2811, Z -7.1667, A 0.000, B 0.000, C 0.000 }
gfCNCPoint5[13200] = {X 5.6885, Y 54.0448, Z -7.1667, A 0.000, B 0.000, C 0.000 }
gfCNCPoint5[13201] = {X 4.7033, Y 53.7614, Z -7.1667, A 0.000, B 0.000, C 0.000 }
gfCNCPoint5[13202] = {X 4.7033, Y 95.2951, Z -7.1667, A 0.000, B 0.000, C 0.000 }
gfCNCPoint5[13203] = {X 117.9387, Y 95.2951, Z -7.1667, A 0.000, B 0.000, C 0.000 }
gfCNCPoint5[13204] = {X 118.3605, Y 94.0800, Z -7.1667, A 0.000, B 0.000, C 0.000 }
gfCNCPoint5[13205] = {X 118.9897, Y 92.9581, Z -7.1667, A 0.000, B 0.000, C 0.000 }
gfCNCPoint5[13206] = {X 119.8064, Y 91.9644, Z -7.1667, A 0.000, B 0.000, C 0.000 }
gfCNCPoint5[13207] = {X 120.7854, Y 91.1300, Z -7.1667, A 0.000, B 0.000, C 0.000 }
gfCNCPoint5[13208] = {X 121.8958, Y 90.4809, Z -7.1667, A 0.000, B 0.000, C 0.000 }
gfCNCPoint5[13209] = {X 123.1032, Y 90.0374, Z -7.1667, A 0.000, B 0.000, C 0.000 }
gfCNCPoint5[13210] = {X 124.3698, Y 89.8133, Z -7.1667, A 0.000, B 0.000, C 0.000 }
gfCNCPoint5[13211] = {X 124.4934, Y 89.7925, Z -7.1667, A 0.000, B 0.000, C 0.000 }
gfCNCPoint5[13212] = {X 125.0314, Y 89.7127, Z -7.1667, A 0.000, B 0.000, C 0.000 }
gfCNCPoint5[13213] = {X 125.3495, Y 89.6657, Z -7.1667, A 0.000, B 0.000, C 0.000 }
gfCNCPoint5[13214] = {X 125.6658, Y 89.6077, Z -7.1667, A 0.000, B 0.000, C 0.000 }
gfCNCPoint5[13215] = {X 126.4580, Y 88.8320, Z -7.1667, A 0.000, B 0.000, C 0.000 }
gfCNCPoint5[13216] = {X 127.2176, Y 88.0243, Z -7.1667, A 0.000, B 0.000, C 0.000 }
gfCNCPoint5[13217] = {X 152.2073, Y 60.5838, Z -7.1667, A 0.000, B 0.000, C 0.000 }
gfCNCPoint5[13218] = {X 152.0684, Y 59.7894, Z -7.1667, A 0.000, B 0.000, C 0.000 }
gfCNCPoint5[13219] = {X 152.0181, Y 58.9845, Z -7.1667, A 0.000, B 0.000, C 0.000 }
gfCNCPoint5[13220] = {X 152.0180, Y 58.0000, Z -7.1667, A 0.000, B 0.000, C 0.000 }
gfCNCPoint5[13221] = {X 152.1286, Y 56.7358, Z -7.1667, A 0.000, B 0.000, C 0.000 }
gfCNCPoint5[13222] = {X 152.4570, Y 55.5101, Z -7.1667, A 0.000, B 0.000, C 0.000 }
gfCNCPoint5[13223] = {X 152.9933, Y 54.3600, Z -7.1667, A 0.000, B 0.000, C 0.000 }
gfCNCPoint5[13224] = {X 153.7212, Y 53.3205, Z -7.1667, A 0.000, B 0.000, C 0.000 }
gfCNCPoint5[13225] = {X 154.6185, Y 52.4232, Z -7.1667, A 0.000, B 0.000, C 0.000 }
gfCNCPoint5[13226] = {X 155.6580, Y 51.6953, Z -7.1667, A 0.000, B 0.000, C 0.000 }
gfCNCPoint5[13227] = {X 156.8081, Y 51.1590, Z -7.1667, A 0.000, B 0.000, C 0.000 }
gfCNCPoint5[13228] = {X 158.0338, Y 50.8306, Z -7.1667, A 0.000, B 0.000, C 0.000 }
gfCNCPoint5[13229] = {X 159.2980, Y 50.7200, Z -7.1667, A 0.000, B 0.000, C 0.000 }
gfCNCPoint5[13230] = {X 178.5335, Y 50.7200, Z -7.1667, A 0.000, B 0.000, C 0.000 }
gfCNCPoint5[13231] = {X 179.7877, Y 50.8289, Z -7.1667, A 0.000, B 0.000, C 0.000 }
gfCNCPoint5[13232] = {X 181.0044, Y 51.1522, Z -7.1667, A 0.000, B 0.000, C 0.000 }
gfCNCPoint5[13233] = {X 182.1472, Y 51.6802, Z -7.1667, A 0.000, B 0.000, C 0.000 }
gfCNCPoint5[13234] = {X 183.1820, Y 52.3973, Z -7.1667, A 0.000, B 0.000, C 0.000 }
gfCNCPoint5[13235] = {X 184.0895, Y 53.2958, Z -7.1667, A 0.000, B 0.000, C 0.000 }
gfCNCPoint5[13236] = {X 184.8260, Y 54.3390, Z -7.1667, A 0.000, B 0.000, C 0.000 }
gfCNCPoint5[13237] = {X 185.3689, Y 55.4949, Z -7.1667, A 0.000, B 0.000, C 0.000 }
gfCNCPoint5[13238] = {X 185.7015, Y 56.7279, Z -7.1667, A 0.000, B 0.000, C 0.000 }
gfCNCPoint5[13239] = {X 185.8135, Y 58.0000, Z -7.1667, A 0.000, B 0.000, C 0.000 }
gfCNCPoint5[13240] = {X 185.8133, Y 58.9942, Z -7.1667, A 0.000, B 0.000, C 0.000 }
gfCNCPoint5[13241] = {X 185.7648, Y 59.7746, Z -7.1667, A 0.000, B 0.000, C 0.000 }
gfCNCPoint5[13242] = {X 185.6330, Y 60.5452, Z -7.1667, A 0.000, B 0.000, C 0.000 }
gfCNCPoint5[13243] = {X 211.4791, Y 88.7602, Z -7.1667, A 0.000, B 0.000, C 0.000 }
gfCNCPoint5[13244] = {X 211.9391, Y 89.2411, Z -7.1667, A 0.000, B 0.000, C 0.000 }
gfCNCPoint5[13245] = {X 212.4193, Y 89.7018, Z -7.1667, A 0.000, B 0.000, C 0.000 }
gfCNCPoint5[13246] = {X 212.5981, Y 89.7394, Z -7.1667, A 0.000, B 0.000, C 0.000 }
gfCNCPoint5[13247] = {X 213.4323, Y 89.8445, Z -7.1667, A 0.000, B 0.000, C 0.000 }
gfCNCPoint5[13248] = {X 214.4196, Y 89.7710, Z -7.1667, A 0.000, B 0.000, C 0.000 }
gfCNCPoint5[13249] = {X 215.4081, Y 89.7159, Z -7.1667, A 0.000, B 0.000, C 0.000 }
gfCNCPoint5[13250] = {X 215.6228, Y 89.6938, Z -7.1667, A 0.000, B 0.000, C 0.000 }
gfCNCPoint5[13251] = {X 215.8202, Y 89.6063, Z -7.1667, A 0.000, B 0.000, C 0.000 }
gfCNCPoint5[13252] = {X 239.3450, Y 74.5358, Z -7.1667, A 0.000, B 0.000, C 0.000 }
gfCNCPoint5[13253] = {X 220.5439, Y 67.1581, Z -7.1667, A 0.000, B 0.000, C 0.000 }
gfCNCPoint5[13254] = {X 219.0948, Y 66.6718, Z -7.1667, A 0.000, B 0.000, C 0.000 }
gfCNCPoint5[13255] = {X 217.5997, Y 66.3543, Z -7.1667, A 0.000, B 0.000, C 0.000 }
gfCNCPoint5[13256] = {X 216.0780, Y 66.2097, Z -7.1667, A 0.000, B 0.000, C 0.000 }
